LIN {X 0,Y 567.569,Z 695.919,A -85,B 0,C 180,E1 -2633.977,E2 -2633.977} C_VEL
LIN {X 0,Y 567.873,Z 675.676,A -85,B 0,C 180,E1 -2636.663,E2 -2636.663} C_VEL
LIN {X 0,Y 568.261,Z 656.786,A -85,B 0,C 180,E1 -2639.242,E2 -2639.242} C_VEL
LIN {X 0,Y 566.233,Z 647.86,A -85,B 0,C 180,E1 -2640.65,E2 -2640.65} C_VEL
LIN {X 0,Y 566.225,Z 647.758,A -85,B 0,C 180,E1 -2643.101,E2 -2643.101} C_VEL
LIN {X 0,Y 566.207,Z 647.757,A -85,B 0,C 180,E1 -2645.688,E2 -2645.688} C_VEL
LIN {X 0,Y 566.21,Z 647.762,A -85,B 0,C 180,E1 -2648.558,E2 -2648.558} C_VEL
LIN {X 0,Y 566.206,Z 647.768,A -85,B 0,C 180,E1 -2651.135,E2 -2651.135} C_VEL
LIN {X 0,Y 566.193,Z 647.762,A -85,B 0,C 180,E1 -2654.035,E2 -2654.035} C_VEL
LIN {X 0,Y 566.208,Z 647.765,A -85,B 0,C 180,E1 -2657.081,E2 -2657.081} C_VEL
LIN {X 0,Y 566.22,Z 647.768,A -85,B 0,C 180,E1 -2659.802,E2 -2659.802} C_VEL
LIN {X 0,Y 566.192,Z 647.763,A -85,B 0,C 180,E1 -2662.598,E2 -2662.598} C_VEL
LIN {X 0,Y 566.214,Z 647.758,A -85,B 0,C 180,E1 -2665.183,E2 -2665.183} C_VEL
LIN {X 0,Y 566.226,Z 647.765,A -85,B 0,C 180,E1 -2667.743,E2 -2667.743} C_VEL
LIN {X 0,Y 566.22,Z 647.758,A -85,B 0,C 180,E1 -2670.322,E2 -2670.322} C_VEL
LIN {X 0,Y 566.226,Z 647.757,A -85,B 0,C 180,E1 -2673.334,E2 -2673.334} C_VEL
LIN {X 0,Y 566.19,Z 647.766,A -85,B 0,C 180,E1 -2675.819,E2 -2675.819} C_VEL
LIN {X 0,Y 566.207,Z 647.766,A -85,B 0,C 180,E1 -2678.902,E2 -2678.902} C_VEL
LIN {X 0,Y 566.203,Z 647.763,A -85,B 0,C 180,E1 -2681.172,E2 -2681.172} C_VEL
LIN {X 0,Y 566.203,Z 647.764,A -85,B 0,C 180,E1 -2684.153,E2 -2684.153} C_VEL
LIN {X 0,Y 566.193,Z 647.766,A -85,B 0,C 180,E1 -2686.359,E2 -2686.359} C_VEL
LIN {X 0,Y 566.264,Z 647.76,A -85,B 0,C 180,E1 -2688.654,E2 -2688.654} C_VEL
LIN {X 0,Y 566.239,Z 647.758,A -85,B 0,C 180,E1 -2691.434,E2 -2691.434} C_VEL
LIN {X 0,Y 566.26,Z 647.755,A -85,B 0,C 180,E1 -2694.302,E2 -2694.302} C_VEL
LIN {X 0,Y 566.271,Z 647.754,A -85,B 0,C 180,E1 -2697.866,E2 -2697.866} C_VEL
LIN {X 0,Y 566.298,Z 647.751,A -85,B 0,C 180,E1 -2700.711,E2 -2700.711} C_VEL
LIN {X 0,Y 566.27,Z 647.752,A -85,B 0,C 180,E1 -2702.845,E2 -2702.845} C_VEL
LIN {X 0,Y 566.26,Z 647.763,A -85,B 0,C 180,E1 -2705.698,E2 -2705.698} C_VEL
LIN {X 0,Y 566.238,Z 647.757,A -85,B 0,C 180,E1 -2708.565,E2 -2708.565} C_VEL
LIN {X 0,Y 566.239,Z 647.762,A -85,B 0,C 180,E1 -2711.454,E2 -2711.454} C_VEL
LIN {X 0,Y 566.222,Z 647.762,A -85,B 0,C 180,E1 -2714.507,E2 -2714.507} C_VEL
LIN {X 0,Y 566.193,Z 647.762,A -85,B 0,C 180,E1 -2717.332,E2 -2717.332} C_VEL
LIN {X 0,Y 566.21,Z 647.769,A -85,B 0,C 180,E1 -2720.337,E2 -2720.337} C_VEL
LIN {X 0,Y 566.219,Z 647.76,A -85,B 0,C 180,E1 -2723.402,E2 -2723.402} C_VEL
LIN {X 0,Y 566.216,Z 647.762,A -85,B 0,C 180,E1 -2725.748,E2 -2725.748} C_VEL
LIN {X 0,Y 566.206,Z 647.757,A -85,B 0,C 180,E1 -2727.492,E2 -2727.492} C_VEL
LIN {X 0,Y 565.528,Z 647.847,A -85,B 0,C 180,E1 -2728.086,E2 -2728.086} C_VEL
LIN {X 0,Y 562.663,Z 648.199,A -85,B 0,C 180,E1 -2729.05,E2 -2729.05} C_VEL
LIN {X 0,Y 560.252,Z 648.499,A -85,B 0,C 180,E1 -2729.825,E2 -2729.825} C_VEL
LIN {X 0,Y 559.223,Z 648.633,A -85,B 0,C 180,E1 -2730.424,E2 -2730.424} C_VEL
LIN {X 0,Y 559.142,Z 648.641,A -85,B 0,C 180,E1 -2730.627,E2 -2730.627} C_VEL
LIN {X 0,Y 559.167,Z 648.638,A -85,B 0,C 180,E1 -2733.574,E2 -2733.574} C_VEL
LIN {X 0,Y 559.159,Z 648.636,A -85,B 0,C 180,E1 -2736.449,E2 -2736.449} C_VEL
LIN {X 0,Y 559.17,Z 648.648,A -85,B 0,C 180,E1 -2738.934,E2 -2738.934} C_VEL
LIN {X 0,Y 559.193,Z 648.637,A -85,B 0,C 180,E1 -2741.767,E2 -2741.767} C_VEL
LIN {X 0,Y 559.131,Z 648.648,A -85,B 0,C 180,E1 -2744.739,E2 -2744.739} C_VEL
LIN {X 0,Y 559.168,Z 648.642,A -85,B 0,C 180,E1 -2747.863,E2 -2747.863} C_VEL
LIN {X 0,Y 559.177,Z 648.639,A -85,B 0,C 180,E1 -2750.135,E2 -2750.135} C_VEL
LIN {X 0,Y 559.139,Z 648.645,A -85,B 0,C 180,E1 -2752.893,E2 -2752.893} C_VEL
LIN {X 0,Y 559.149,Z 648.651,A -85,B 0,C 180,E1 -2755.556,E2 -2755.556} C_VEL
LIN {X 0,Y 559.165,Z 648.643,A -85,B 0,C 180,E1 -2758.138,E2 -2758.138} C_VEL
LIN {X 0,Y 559.15,Z 648.642,A -85,B 0,C 180,E1 -2760.648,E2 -2760.648} C_VEL
LIN {X 0,Y 559.166,Z 648.641,A -85,B 0,C 180,E1 -2763.172,E2 -2763.172} C_VEL
LIN {X 0,Y 559.152,Z 648.644,A -85,B 0,C 180,E1 -2765.495,E2 -2765.495} C_VEL
LIN {X 0,Y 559.166,Z 648.643,A -85,B 0,C 180,E1 -2768.624,E2 -2768.624} C_VEL
LIN {X 0,Y 559.164,Z 648.641,A -85,B 0,C 180,E1 -2770.927,E2 -2770.927} C_VEL
LIN {X 0,Y 559.163,Z 648.644,A -85,B 0,C 180,E1 -2773.948,E2 -2773.948} C_VEL
LIN {X 0,Y 559.168,Z 648.646,A -85,B 0,C 180,E1 -2776.184,E2 -2776.184} C_VEL
LIN {X 0,Y 559.191,Z 648.639,A -85,B 0,C 180,E1 -2779.134,E2 -2779.134} C_VEL
LIN {X 0,Y 559.202,Z 648.637,A -85,B 0,C 180,E1 -2782.054,E2 -2782.054} C_VEL
LIN {X 0,Y 559.25,Z 648.638,A -85,B 0,C 180,E1 -2784.953,E2 -2784.953} C_VEL
LIN {X 0,Y 559.25,Z 648.629,A -85,B 0,C 180,E1 -2787.839,E2 -2787.839} C_VEL
LIN {X 0,Y 559.268,Z 648.633,A -85,B 0,C 180,E1 -2790.72,E2 -2790.72} C_VEL
LIN {X 0,Y 559.235,Z 648.638,A -85,B 0,C 180,E1 -2792.881,E2 -2792.881} C_VEL
LIN {X 0,Y 559.226,Z 648.635,A -85,B 0,C 180,E1 -2795.77,E2 -2795.77} C_VEL
LIN {X 0,Y 559.188,Z 648.639,A -85,B 0,C 180,E1 -2798.674,E2 -2798.674} C_VEL
LIN {X 0,Y 559.201,Z 648.644,A -85,B 0,C 180,E1 -2801.6,E2 -2801.6} C_VEL
LIN {X 0,Y 559.195,Z 648.637,A -85,B 0,C 180,E1 -2804.595,E2 -2804.595} C_VEL
LIN {X 0,Y 559.155,Z 648.649,A -85,B 0,C 180,E1 -2807.557,E2 -2807.557} C_VEL
LIN {X 0,Y 559.167,Z 648.65,A -85,B 0,C 180,E1 -2809.837,E2 -2809.837} C_VEL
LIN {X 0,Y 559.136,Z 648.65,A -85,B 0,C 180,E1 -2812.152,E2 -2812.152} C_VEL
LIN {X 0,Y 559.173,Z 648.639,A -85,B 0,C 180,E1 -2815.187,E2 -2815.187} C_VEL
LIN {X 0,Y 559.187,Z 648.641,A -85,B 0,C 180,E1 -2817.711,E2 -2817.711} C_VEL
LIN {X 0,Y 559.162,Z 648.65,A -85,B 0,C 180,E1 -2820.181,E2 -2820.181} C_VEL
LIN {X 0,Y 559.169,Z 648.644,A -85,B 0,C 180,E1 -2822.713,E2 -2822.713} C_VEL
LIN {X 0,Y 559.15,Z 648.642,A -85,B 0,C 180,E1 -2825.321,E2 -2825.321} C_VEL
LIN {X 0,Y 559.127,Z 648.647,A -85,B 0,C 180,E1 -2828.017,E2 -2828.017} C_VEL
LIN {X 0,Y 559.168,Z 648.648,A -85,B 0,C 180,E1 -2830.81,E2 -2830.81} C_VEL
LIN {X 0,Y 559.135,Z 648.643,A -85,B 0,C 180,E1 -2833.733,E2 -2833.733} C_VEL
LIN {X 0,Y 559.164,Z 648.649,A -85,B 0,C 180,E1 -2836.8,E2 -2836.8} C_VEL
LIN {X 0,Y 559.171,Z 648.646,A -85,B 0,C 180,E1 -2839.189,E2 -2839.189} C_VEL
LIN {X 0,Y 559.126,Z 648.642,A -85,B 0,C 180,E1 -2841.982,E2 -2841.982} C_VEL
LIN {X 0,Y 559.151,Z 648.637,A -85,B 0,C 180,E1 -2844.782,E2 -2844.782} C_VEL
LIN {X 0,Y 559.164,Z 648.65,A -85,B 0,C 180,E1 -2847.361,E2 -2847.361} C_VEL
LIN {X 0,Y 559.179,Z 648.631,A -85,B 0,C 180,E1 -2850.135,E2 -2850.135} C_VEL
LIN {X 0,Y 559.171,Z 648.637,A -85,B 0,C 180,E1 -2853.17,E2 -2853.17} C_VEL
LIN {X 0,Y 559.15,Z 648.649,A -85,B 0,C 180,E1 -2855.495,E2 -2855.495} C_VEL
LIN {X 0,Y 559.153,Z 648.641,A -85,B 0,C 180,E1 -2858.447,E2 -2858.447} C_VEL
LIN {X 0,Y 559.161,Z 648.639,A -85,B 0,C 180,E1 -2860.926,E2 -2860.926} C_VEL
LIN {X 0,Y 559.162,Z 648.648,A -85,B 0,C 180,E1 -2863.948,E2 -2863.948} C_VEL
LIN {X 0,Y 559.164,Z 648.644,A -85,B 0,C 180,E1 -2866.184,E2 -2866.184} C_VEL
LIN {X 0,Y 559.201,Z 648.634,A -85,B 0,C 180,E1 -2869.134,E2 -2869.134} C_VEL
LIN {X 0,Y 559.203,Z 648.638,A -85,B 0,C 180,E1 -2872.054,E2 -2872.054} C_VEL
LIN {X 0,Y 559.252,Z 648.631,A -85,B 0,C 180,E1 -2874.954,E2 -2874.954} C_VEL
LIN {X 0,Y 559.242,Z 648.627,A -85,B 0,C 180,E1 -2877.84,E2 -2877.84} C_VEL
LIN {X 0,Y 559.269,Z 648.635,A -85,B 0,C 180,E1 -2880.72,E2 -2880.72} C_VEL
LIN {X 0,Y 559.236,Z 648.637,A -85,B 0,C 180,E1 -2882.882,E2 -2882.882} C_VEL
LIN {X 0,Y 559.229,Z 648.631,A -85,B 0,C 180,E1 -2885.77,E2 -2885.77} C_VEL
LIN {X 0,Y 559.194,Z 648.636,A -85,B 0,C 180,E1 -2888.674,E2 -2888.674} C_VEL
LIN {X 0,Y 559.198,Z 648.636,A -85,B 0,C 180,E1 -2891.601,E2 -2891.601} C_VEL
LIN {X 0,Y 559.188,Z 648.636,A -85,B 0,C 180,E1 -2894.596,E2 -2894.596} C_VEL
LIN {X 0,Y 559.154,Z 648.646,A -85,B 0,C 180,E1 -2897.557,E2 -2897.557} C_VEL
LIN {X 0,Y 559.165,Z 648.643,A -85,B 0,C 180,E1 -2899.838,E2 -2899.838} C_VEL
LIN {X 0,Y 559.134,Z 648.642,A -85,B 0,C 180,E1 -2902.153,E2 -2902.153} C_VEL
LIN {X 0,Y 559.17,Z 648.642,A -85,B 0,C 180,E1 -2905.188,E2 -2905.188} C_VEL
LIN {X 0,Y 559.185,Z 648.637,A -85,B 0,C 180,E1 -2907.712,E2 -2907.712} C_VEL
LIN {X 0,Y 559.16,Z 648.643,A -85,B 0,C 180,E1 -2910.182,E2 -2910.182} C_VEL
LIN {X 0,Y 559.167,Z 648.64,A -85,B 0,C 180,E1 -2912.715,E2 -2912.715} C_VEL
LIN {X 0,Y 559.151,Z 648.637,A -85,B 0,C 180,E1 -2915.322,E2 -2915.322} C_VEL
LIN {X 0,Y 559.129,Z 648.65,A -85,B 0,C 180,E1 -2918.018,E2 -2918.018} C_VEL
LIN {X 0,Y 559.173,Z 648.636,A -85,B 0,C 180,E1 -2920.811,E2 -2920.811} C_VEL
LIN {X 0,Y 559.158,Z 648.642,A -85,B 0,C 180,E1 -2923.732,E2 -2923.732} C_VEL
LIN {X 0,Y 559.161,Z 648.647,A -85,B 0,C 180,E1 -2926.802,E2 -2926.802} C_VEL
LIN {X 0,Y 559.171,Z 648.641,A -85,B 0,C 180,E1 -2929.19,E2 -2929.19} C_VEL
LIN {X 0,Y 559.13,Z 648.644,A -85,B 0,C 180,E1 -2931.983,E2 -2931.983} C_VEL
LIN {X 0,Y 559.154,Z 648.642,A -85,B 0,C 180,E1 -2934.784,E2 -2934.784} C_VEL
LIN {X 0,Y 559.171,Z 648.628,A -85,B 0,C 180,E1 -2937.362,E2 -2937.362} C_VEL
LIN {X 0,Y 559.219,Z 648.853,A -85,B 0,C 180,E1 -2939.09,E2 -2939.09} C_VEL
LIN {X 0,Y 561.438,Z 658.244,A -85,B 0,C 180,E1 -2940.573,E2 -2940.573} C_VEL
LIN {X 0,Y 561.129,Z 674.15,A -85,B 0,C 180,E1 -2942.78,E2 -2942.78} C_VEL
LIN {X 0,Y 560.756,Z 691.767,A -85,B 0,C 180,E1 -2945.175,E2 -2945.175} C_VEL
LIN {X 0,Y 560.706,Z 696.007,A -85,B 0,C 180,E1 -2945.716,E2 -2945.716} C_VEL
LIN {X 0,Y 563.185,Z 706.581,A -85,B 0,C 180,E1 -2945.992,E2 -2945.992} C_VEL
LIN {X 0,Y 562.287,Z 897.325,A -85,B 0,C 180,E1 -2948.556,E2 -2948.556} C_VEL
LIN {X 0,Y 562.123,Z 911.373,A -85,B 0,C 180,E1 -2948.838,E2 -2948.838} C_VEL
LIN {X 0,Y 561.91,Z 924.892,A -85,B 0,C 180,E1 -2949.214,E2 -2949.214} C_VEL
LIN {X 0,Y 561.684,Z 938.18,A -85,B 0,C 180,E1 -2949.684,E2 -2949.684} C_VEL
LIN {X 0,Y 561.381,Z 951.016,A -85,B 0,C 180,E1 -2950.244,E2 -2950.244} C_VEL
LIN {X 0,Y 561.089,Z 963.63,A -85,B 0,C 180,E1 -2950.9,E2 -2950.9} C_VEL
LIN {X 0,Y 560.713,Z 977.24,A -85,B 0,C 180,E1 -2951.739,E2 -2951.739} C_VEL
LIN {X 0,Y 560.337,Z 992.413,A -85,B 0,C 180,E1 -2952.858,E2 -2952.858} C_VEL
LIN {X 0,Y 559.998,Z 1005.074,A -85,B 0,C 180,E1 -2953.973,E2 -2953.973} C_VEL
LIN {X 0,Y 559.712,Z 1015.89,A -85,B 0,C 180,E1 -2955.077,E2 -2955.077} C_VEL
LIN {X 0,Y 559.449,Z 1026.869,A -85,B 0,C 180,E1 -2956.377,E2 -2956.377} C_VEL
LIN {X 0,Y 559.241,Z 1036.211,A -85,B 0,C 180,E1 -2957.665,E2 -2957.665} C_VEL
LIN {X 0,Y 559.063,Z 1045.284,A -85,B 0,C 180,E1 -2959.131,E2 -2959.131} C_VEL
LIN {X 0,Y 558.941,Z 1052.854,A -85,B 0,C 180,E1 -2960.593,E2 -2960.593} C_VEL
LIN {X 0,Y 558.89,Z 1059.068,A -85,B 0,C 180,E1 -2962.049,E2 -2962.049} C_VEL
LIN {X 0,Y 558.841,Z 1064.1,A -85,B 0,C 180,E1 -2963.501,E2 -2963.501} C_VEL
LIN {X 0,Y 558.776,Z 1068.061,A -85,B 0,C 180,E1 -2964.949,E2 -2964.949} C_VEL
LIN {X 0,Y 558.817,Z 1070.961,A -85,B 0,C 180,E1 -2966.395,E2 -2966.395} C_VEL
LIN {X 0,Y 558.734,Z 1072.881,A -85,B 0,C 180,E1 -2967.837,E2 -2967.837} C_VEL
LIN {X 0,Y 558.738,Z 1073.833,A -85,B 0,C 180,E1 -2969.279,E2 -2969.279} C_VEL
LIN {X 0,Y 558.738,Z 1073.833,A -85,B 0,C 180,E1 -2970.721,E2 -2970.721} C_VEL
LIN {X 0,Y 558.734,Z 1072.881,A -85,B 0,C 180,E1 -2972.163,E2 -2972.163} C_VEL
LIN {X 0,Y 558.817,Z 1070.961,A -85,B 0,C 180,E1 -2973.605,E2 -2973.605} C_VEL
LIN {X 0,Y 558.776,Z 1068.061,A -85,B 0,C 180,E1 -2975.051,E2 -2975.051} C_VEL
LIN {X 0,Y 558.841,Z 1063.992,A -85,B 0,C 180,E1 -2976.535,E2 -2976.535} C_VEL
LIN {X 0,Y 558.89,Z 1059.068,A -85,B 0,C 180,E1 -2977.951,E2 -2977.951} C_VEL
LIN {X 0,Y 558.941,Z 1052.854,A -85,B 0,C 180,E1 -2979.407,E2 -2979.407} C_VEL
LIN {X 0,Y 559.115,Z 1044.27,A -85,B 0,C 180,E1 -2981.046,E2 -2981.046} C_VEL
LIN {X 0,Y 559.241,Z 1036.211,A -85,B 0,C 180,E1 -2982.335,E2 -2982.335} C_VEL
LIN {X 0,Y 559.449,Z 1026.869,A -85,B 0,C 180,E1 -2983.623,E2 -2983.623} C_VEL
LIN {X 0,Y 559.71,Z 1015.898,A -85,B 0,C 180,E1 -2984.923,E2 -2984.923} C_VEL
LIN {X 0,Y 559.975,Z 1005.074,A -85,B 0,C 180,E1 -2986.028,E2 -2986.028} C_VEL
LIN {X 0,Y 560.341,Z 991.252,A -85,B 0,C 180,E1 -2987.236,E2 -2987.236} C_VEL
LIN {X 0,Y 560.713,Z 977.24,A -85,B 0,C 180,E1 -2988.261,E2 -2988.261} C_VEL
LIN {X 0,Y 561.087,Z 963.63,A -85,B 0,C 180,E1 -2989.1,E2 -2989.1} C_VEL
LIN {X 0,Y 561.37,Z 951.016,A -85,B 0,C 180,E1 -2989.756,E2 -2989.756} C_VEL
LIN {X 0,Y 561.701,Z 936.508,A -85,B 0,C 180,E1 -2990.382,E2 -2990.382} C_VEL
LIN {X 0,Y 561.995,Z 921.141,A -85,B 0,C 180,E1 -2990.903,E2 -2990.903} C_VEL
LIN {X 0,Y 562.224,Z 902.928,A -85,B 0,C 180,E1 -2991.35,E2 -2991.35} C_VEL
LIN {X 0,Y 562.457,Z 877.103,A -85,B 0,C 180,E1 -2991.725,E2 -2991.725} C_VEL
LIN {X 0,Y 563.09,Z 705.526,A -85,B 0,C 180,E1 -2994.026,E2 -2994.026} C_VEL
LIN {X 0,Y 560.696,Z 695.906,A -85,B 0,C 180,E1 -2994.29,E2 -2994.29} C_VEL
LIN {X 0,Y 561.115,Z 676.134,A -85,B 0,C 180,E1 -2996.947,E2 -2996.947} C_VEL
LIN {X 0,Y 561.522,Z 659.701,A -85,B 0,C 180,E1 -2999.216,E2 -2999.216} C_VEL
LIN {X 0,Y 560.763,Z 655.01,A -85,B 0,C 180,E1 -2999.924,E2 -2999.924} C_VEL
LIN {X 0,Y 559.214,Z 648.775,A -85,B 0,C 180,E1 -3000.936,E2 -3000.936} C_VEL
LIN {X 0,Y 559.163,Z 648.643,A -85,B 0,C 180,E1 -3003.949,E2 -3003.949} C_VEL
LIN {X 0,Y 559.164,Z 648.63,A -85,B 0,C 180,E1 -3006.448,E2 -3006.448} C_VEL
LIN {X 0,Y 559.173,Z 648.642,A -85,B 0,C 180,E1 -3008.933,E2 -3008.933} C_VEL
LIN {X 0,Y 559.186,Z 648.642,A -85,B 0,C 180,E1 -3011.767,E2 -3011.767} C_VEL
LIN {X 0,Y 559.133,Z 648.639,A -85,B 0,C 180,E1 -3014.738,E2 -3014.738} C_VEL
LIN {X 0,Y 559.167,Z 648.644,A -85,B 0,C 180,E1 -3017.257,E2 -3017.257} C_VEL
LIN {X 0,Y 559.18,Z 648.642,A -85,B 0,C 180,E1 -3020.135,E2 -3020.135} C_VEL
LIN {X 0,Y 559.139,Z 648.641,A -85,B 0,C 180,E1 -3022.892,E2 -3022.892} C_VEL
LIN {X 0,Y 559.155,Z 648.64,A -85,B 0,C 180,E1 -3025.556,E2 -3025.556} C_VEL
LIN {X 0,Y 559.163,Z 648.647,A -85,B 0,C 180,E1 -3028.137,E2 -3028.137} C_VEL
LIN {X 0,Y 559.15,Z 648.632,A -85,B 0,C 180,E1 -3030.647,E2 -3030.647} C_VEL
LIN {X 0,Y 559.173,Z 648.635,A -85,B 0,C 180,E1 -3033.169,E2 -3033.169} C_VEL
LIN {X 0,Y 559.147,Z 648.642,A -85,B 0,C 180,E1 -3035.494,E2 -3035.494} C_VEL
LIN {X 0,Y 559.167,Z 648.648,A -85,B 0,C 180,E1 -3038.624,E2 -3038.624} C_VEL
LIN {X 0,Y 559.162,Z 648.642,A -85,B 0,C 180,E1 -3040.926,E2 -3040.926} C_VEL
LIN {X 0,Y 559.165,Z 648.639,A -85,B 0,C 180,E1 -3043.948,E2 -3043.948} C_VEL
LIN {X 0,Y 559.165,Z 648.64,A -85,B 0,C 180,E1 -3046.184,E2 -3046.184} C_VEL
LIN {X 0,Y 559.223,Z 648.639,A -85,B 0,C 180,E1 -3049.134,E2 -3049.134} C_VEL
LIN {X 0,Y 559.203,Z 648.63,A -85,B 0,C 180,E1 -3052.053,E2 -3052.053} C_VEL
LIN {X 0,Y 559.252,Z 648.635,A -85,B 0,C 180,E1 -3054.953,E2 -3054.953} C_VEL
LIN {X 0,Y 559.242,Z 648.63,A -85,B 0,C 180,E1 -3057.839,E2 -3057.839} C_VEL
LIN {X 0,Y 559.268,Z 648.627,A -85,B 0,C 180,E1 -3060.72,E2 -3060.72} C_VEL
LIN {X 0,Y 559.236,Z 648.628,A -85,B 0,C 180,E1 -3062.881,E2 -3062.881} C_VEL
LIN {X 0,Y 559.229,Z 648.638,A -85,B 0,C 180,E1 -3065.77,E2 -3065.77} C_VEL
LIN {X 0,Y 559.193,Z 648.634,A -85,B 0,C 180,E1 -3068.674,E2 -3068.674} C_VEL
LIN {X 0,Y 559.197,Z 648.642,A -85,B 0,C 180,E1 -3071.6,E2 -3071.6} C_VEL
LIN {X 0,Y 559.187,Z 648.638,A -85,B 0,C 180,E1 -3074.596,E2 -3074.596} C_VEL
LIN {X 0,Y 559.153,Z 648.641,A -85,B 0,C 180,E1 -3077.557,E2 -3077.557} C_VEL
LIN {X 0,Y 559.164,Z 648.644,A -85,B 0,C 180,E1 -3079.837,E2 -3079.837} C_VEL
LIN {X 0,Y 559.145,Z 648.649,A -85,B 0,C 180,E1 -3082.152,E2 -3082.152} C_VEL
LIN {X 0,Y 559.15,Z 648.649,A -85,B 0,C 180,E1 -3084.505,E2 -3084.505} C_VEL
LIN {X 0,Y 559.169,Z 648.636,A -85,B 0,C 180,E1 -3086.902,E2 -3086.902} C_VEL
LIN {X 0,Y 559.179,Z 648.631,A -85,B 0,C 180,E1 -3089.865,E2 -3089.865} C_VEL
LIN {X 0,Y 559.142,Z 648.641,A -85,B 0,C 180,E1 -3090.627,E2 -3090.627} C_VEL
LIN {X 0,Y 558.479,Z 648.728,A -85,B 0,C 180,E1 -3091.228,E2 -3091.228} C_VEL
LIN {X 0,Y 555.616,Z 649.084,A -85,B 0,C 180,E1 -3092.204,E2 -3092.204} C_VEL
LIN {X 0,Y 553.205,Z 649.387,A -85,B 0,C 180,E1 -3092.99,E2 -3092.99} C_VEL
LIN {X 0,Y 552.187,Z 649.508,A -85,B 0,C 180,E1 -3093.597,E2 -3093.597} C_VEL
LIN {X 0,Y 552.113,Z 649.517,A -85,B 0,C 180,E1 -3093.802,E2 -3093.802} C_VEL
LIN {X 0,Y 552.102,Z 649.517,A -85,B 0,C 180,E1 -3096.747,E2 -3096.747} C_VEL
LIN {X 0,Y 552.126,Z 649.519,A -85,B 0,C 180,E1 -3099.527,E2 -3099.527} C_VEL
LIN {X 0,Y 552.163,Z 649.516,A -85,B 0,C 180,E1 -3101.441,E2 -3101.441} C_VEL
LIN {X 0,Y 552.087,Z 649.523,A -85,B 0,C 180,E1 -3104.532,E2 -3104.532} C_VEL
LIN {X 0,Y 552.122,Z 649.523,A -85,B 0,C 180,E1 -3107.585,E2 -3107.585} C_VEL
LIN {X 0,Y 552.126,Z 649.517,A -85,B 0,C 180,E1 -3110.474,E2 -3110.474} C_VEL
LIN {X 0,Y 552.114,Z 649.526,A -85,B 0,C 180,E1 -3113.315,E2 -3113.315} C_VEL
LIN {X 0,Y 552.124,Z 649.523,A -85,B 0,C 180,E1 -3115.94,E2 -3115.94} C_VEL
LIN {X 0,Y 552.112,Z 649.519,A -85,B 0,C 180,E1 -3118.541,E2 -3118.541} C_VEL
LIN {X 0,Y 552.119,Z 649.522,A -85,B 0,C 180,E1 -3121.438,E2 -3121.438} C_VEL
LIN {X 0,Y 552.125,Z 649.521,A -85,B 0,C 180,E1 -3124.356,E2 -3124.356} C_VEL
LIN {X 0,Y 552.105,Z 649.521,A -85,B 0,C 180,E1 -3126.759,E2 -3126.759} C_VEL
LIN {X 0,Y 552.115,Z 649.518,A -85,B 0,C 180,E1 -3129.12,E2 -3129.12} C_VEL
LIN {X 0,Y 552.121,Z 649.518,A -85,B 0,C 180,E1 -3131.445,E2 -3131.445} C_VEL
LIN {X 0,Y 552.112,Z 649.52,A -85,B 0,C 180,E1 -3133.738,E2 -3133.738} C_VEL
LIN {X 0,Y 552.132,Z 649.521,A -85,B 0,C 180,E1 -3136.005,E2 -3136.005} C_VEL
LIN {X 0,Y 552.158,Z 649.517,A -85,B 0,C 180,E1 -3138.994,E2 -3138.994} C_VEL
LIN {X 0,Y 552.156,Z 649.514,A -85,B 0,C 180,E1 -3141.952,E2 -3141.952} C_VEL
LIN {X 0,Y 552.225,Z 649.513,A -85,B 0,C 180,E1 -3144.889,E2 -3144.889} C_VEL
LIN {X 0,Y 552.221,Z 649.505,A -85,B 0,C 180,E1 -3147.812,E2 -3147.812} C_VEL
LIN {X 0,Y 552.238,Z 649.509,A -85,B 0,C 180,E1 -3150.729,E2 -3150.729} C_VEL
LIN {X 0,Y 552.202,Z 649.515,A -85,B 0,C 180,E1 -3152.918,E2 -3152.918} C_VEL
LIN {X 0,Y 552.196,Z 649.51,A -85,B 0,C 180,E1 -3155.844,E2 -3155.844} C_VEL
LIN {X 0,Y 552.158,Z 649.515,A -85,B 0,C 180,E1 -3158.785,E2 -3158.785} C_VEL
LIN {X 0,Y 552.159,Z 649.519,A -85,B 0,C 180,E1 -3161.75,E2 -3161.75} C_VEL
LIN {X 0,Y 552.132,Z 649.517,A -85,B 0,C 180,E1 -3164.748,E2 -3164.748} C_VEL
LIN {X 0,Y 552.106,Z 649.528,A -85,B 0,C 180,E1 -3167.788,E2 -3167.788} C_VEL
LIN {X 0,Y 552.126,Z 649.523,A -85,B 0,C 180,E1 -3170.101,E2 -3170.101} C_VEL
LIN {X 0,Y 552.091,Z 649.524,A -85,B 0,C 180,E1 -3172.45,E2 -3172.45} C_VEL
LIN {X 0,Y 552.15,Z 649.515,A -85,B 0,C 180,E1 -3175.35,E2 -3175.35} C_VEL
LIN {X 0,Y 552.12,Z 649.527,A -85,B 0,C 180,E1 -3178.097,E2 -3178.097} C_VEL
LIN {X 0,Y 552.108,Z 649.524,A -85,B 0,C 180,E1 -3180.608,E2 -3180.608} C_VEL
LIN {X 0,Y 552.116,Z 649.519,A -85,B 0,C 180,E1 -3183.185,E2 -3183.185} C_VEL
LIN {X 0,Y 552.105,Z 649.521,A -85,B 0,C 180,E1 -3185.841,E2 -3185.841} C_VEL
LIN {X 0,Y 552.117,Z 649.521,A -85,B 0,C 180,E1 -3189.061,E2 -3189.061} C_VEL
LIN {X 0,Y 552.131,Z 649.517,A -85,B 0,C 180,E1 -3191.444,E2 -3191.444} C_VEL
LIN {X 0,Y 552.087,Z 649.528,A -85,B 0,C 180,E1 -3194.532,E2 -3194.532} C_VEL
LIN {X 0,Y 552.123,Z 649.518,A -85,B 0,C 180,E1 -3197.584,E2 -3197.584} C_VEL
LIN {X 0,Y 552.134,Z 649.516,A -85,B 0,C 180,E1 -3199.792,E2 -3199.792} C_VEL
LIN {X 0,Y 552.084,Z 649.52,A -85,B 0,C 180,E1 -3202.336,E2 -3202.336} C_VEL
LIN {X 0,Y 552.122,Z 649.516,A -85,B 0,C 180,E1 -3205.054,E2 -3205.054} C_VEL
LIN {X 0,Y 552.118,Z 649.522,A -85,B 0,C 180,E1 -3207.682,E2 -3207.682} C_VEL
LIN {X 0,Y 552.135,Z 649.507,A -85,B 0,C 180,E1 -3210.237,E2 -3210.237} C_VEL
LIN {X 0,Y 552.136,Z 649.511,A -85,B 0,C 180,E1 -3212.998,E2 -3212.998} C_VEL
LIN {X 0,Y 552.104,Z 649.522,A -85,B 0,C 180,E1 -3215.161,E2 -3215.161} C_VEL
LIN {X 0,Y 552.104,Z 649.525,A -85,B 0,C 180,E1 -3217.55,E2 -3217.55} C_VEL
LIN {X 0,Y 552.146,Z 649.513,A -85,B 0,C 180,E1 -3220.674,E2 -3220.674} C_VEL
LIN {X 0,Y 552.111,Z 649.522,A -85,B 0,C 180,E1 -3223.737,E2 -3223.737} C_VEL
LIN {X 0,Y 552.126,Z 649.525,A -85,B 0,C 180,E1 -3226.005,E2 -3226.005} C_VEL
LIN {X 0,Y 552.168,Z 649.511,A -85,B 0,C 180,E1 -3228.994,E2 -3228.994} C_VEL
LIN {X 0,Y 552.156,Z 649.515,A -85,B 0,C 180,E1 -3231.952,E2 -3231.952} C_VEL
LIN {X 0,Y 552.227,Z 649.507,A -85,B 0,C 180,E1 -3234.889,E2 -3234.889} C_VEL
LIN {X 0,Y 552.214,Z 649.502,A -85,B 0,C 180,E1 -3237.812,E2 -3237.812} C_VEL
LIN {X 0,Y 552.239,Z 649.511,A -85,B 0,C 180,E1 -3240.729,E2 -3240.729} C_VEL
LIN {X 0,Y 552.202,Z 649.513,A -85,B 0,C 180,E1 -3242.918,E2 -3242.918} C_VEL
LIN {X 0,Y 552.199,Z 649.507,A -85,B 0,C 180,E1 -3245.844,E2 -3245.844} C_VEL
LIN {X 0,Y 552.162,Z 649.513,A -85,B 0,C 180,E1 -3248.786,E2 -3248.786} C_VEL
LIN {X 0,Y 552.154,Z 649.512,A -85,B 0,C 180,E1 -3251.751,E2 -3251.751} C_VEL
LIN {X 0,Y 552.126,Z 649.518,A -85,B 0,C 180,E1 -3254.749,E2 -3254.749} C_VEL
LIN {X 0,Y 552.105,Z 649.52,A -85,B 0,C 180,E1 -3257.789,E2 -3257.789} C_VEL
LIN {X 0,Y 552.124,Z 649.518,A -85,B 0,C 180,E1 -3260.102,E2 -3260.102} C_VEL
LIN {X 0,Y 552.088,Z 649.518,A -85,B 0,C 180,E1 -3262.451,E2 -3262.451} C_VEL
LIN {X 0,Y 552.147,Z 649.519,A -85,B 0,C 180,E1 -3265.352,E2 -3265.352} C_VEL
LIN {X 0,Y 552.118,Z 649.509,A -85,B 0,C 180,E1 -3268.098,E2 -3268.098} C_VEL
LIN {X 0,Y 552.105,Z 649.517,A -85,B 0,C 180,E1 -3270.609,E2 -3270.609} C_VEL
LIN {X 0,Y 552.121,Z 649.517,A -85,B 0,C 180,E1 -3273.185,E2 -3273.185} C_VEL
LIN {X 0,Y 552.106,Z 649.519,A -85,B 0,C 180,E1 -3275.842,E2 -3275.842} C_VEL
LIN {X 0,Y 552.12,Z 649.517,A -85,B 0,C 180,E1 -3279.063,E2 -3279.063} C_VEL
LIN {X 0,Y 552.165,Z 649.506,A -85,B 0,C 180,E1 -3281.442,E2 -3281.442} C_VEL
LIN {X 0,Y 552.09,Z 649.525,A -85,B 0,C 180,E1 -3284.533,E2 -3284.533} C_VEL
LIN {X 0,Y 552.125,Z 649.517,A -85,B 0,C 180,E1 -3287.585,E2 -3287.585} C_VEL
LIN {X 0,Y 552.129,Z 649.523,A -85,B 0,C 180,E1 -3290.474,E2 -3290.474} C_VEL
LIN {X 0,Y 552.11,Z 649.507,A -85,B 0,C 180,E1 -3293.316,E2 -3293.316} C_VEL
LIN {X 0,Y 552.127,Z 649.52,A -85,B 0,C 180,E1 -3295.94,E2 -3295.94} C_VEL
LIN {X 0,Y 552.128,Z 649.643,A -85,B 0,C 180,E1 -3298.782,E2 -3298.782} C_VEL
LIN {X 0,Y 554.588,Z 659.655,A -85,B 0,C 180,E1 -3300.382,E2 -3300.382} C_VEL
LIN {X 0,Y 554.665,Z 665.531,A -85,B 0,C 180,E1 -3301.218,E2 -3301.218} C_VEL
LIN {X 0,Y 554.098,Z 687.223,A -85,B 0,C 180,E1 -3304.229,E2 -3304.229} C_VEL
LIN {X 0,Y 553.914,Z 695.92,A -85,B 0,C 180,E1 -3305.393,E2 -3305.393} C_VEL
LIN {X 0,Y 556.651,Z 707.052,A -85,B 0,C 180,E1 -3305.699,E2 -3305.699} C_VEL
LIN {X 0,Y 555.74,Z 894.458,A -85,B 0,C 180,E1 -3308.242,E2 -3308.242} C_VEL
LIN {X 0,Y 555.514,Z 909.386,A -85,B 0,C 180,E1 -3308.525,E2 -3308.525} C_VEL
LIN {X 0,Y 555.284,Z 924.13,A -85,B 0,C 180,E1 -3308.93,E2 -3308.93} C_VEL
LIN {X 0,Y 555.002,Z 937.152,A -85,B 0,C 180,E1 -3309.388,E2 -3309.388} C_VEL
LIN {X 0,Y 554.715,Z 949.907,A -85,B 0,C 180,E1 -3309.943,E2 -3309.943} C_VEL
LIN {X 0,Y 554.368,Z 961.945,A -85,B 0,C 180,E1 -3310.563,E2 -3310.563} C_VEL
LIN {X 0,Y 553.989,Z 974.377,A -85,B 0,C 180,E1 -3311.318,E2 -3311.318} C_VEL
LIN {X 0,Y 553.644,Z 986.62,A -85,B 0,C 180,E1 -3312.186,E2 -3312.186} C_VEL
LIN {X 0,Y 553.263,Z 998.97,A -85,B 0,C 180,E1 -3313.203,E2 -3313.203} C_VEL
LIN {X 0,Y 552.928,Z 1010.762,A -85,B 0,C 180,E1 -3314.33,E2 -3314.33} C_VEL
LIN {X 0,Y 552.561,Z 1023.939,A -85,B 0,C 180,E1 -3315.828,E2 -3315.828} C_VEL
LIN {X 0,Y 552.272,Z 1033.679,A -85,B 0,C 180,E1 -3317.133,E2 -3317.133} C_VEL
LIN {X 0,Y 552.125,Z 1040.927,A -85,B 0,C 180,E1 -3318.249,E2 -3318.249} C_VEL
LIN {X 0,Y 551.974,Z 1049.198,A -85,B 0,C 180,E1 -3319.732,E2 -3319.732} C_VEL
LIN {X 0,Y 551.855,Z 1056.075,A -85,B 0,C 180,E1 -3321.21,E2 -3321.21} C_VEL
LIN {X 0,Y 551.808,Z 1061.739,A -85,B 0,C 180,E1 -3322.683,E2 -3322.683} C_VEL
LIN {X 0,Y 551.77,Z 1066.23,A -85,B 0,C 180,E1 -3324.152,E2 -3324.152} C_VEL
LIN {X 0,Y 551.701,Z 1069.655,A -85,B 0,C 180,E1 -3325.617,E2 -3325.617} C_VEL
LIN {X 0,Y 551.712,Z 1072.084,A -85,B 0,C 180,E1 -3327.079,E2 -3327.079} C_VEL
LIN {X 0,Y 551.64,Z 1073.499,A -85,B 0,C 180,E1 -3328.54,E2 -3328.54} C_VEL
LIN {X 0,Y 551.636,Z 1074,A -85,B 0,C 180,E1 -3330,E2 -3330} C_VEL
LIN {X 0,Y 551.64,Z 1073.499,A -85,B 0,C 180,E1 -3331.46,E2 -3331.46} C_VEL
LIN {X 0,Y 551.712,Z 1072.084,A -85,B 0,C 180,E1 -3332.921,E2 -3332.921} C_VEL
LIN {X 0,Y 551.702,Z 1069.655,A -85,B 0,C 180,E1 -3334.383,E2 -3334.383} C_VEL
LIN {X 0,Y 551.769,Z 1066.23,A -85,B 0,C 180,E1 -3335.848,E2 -3335.848} C_VEL
LIN {X 0,Y 551.808,Z 1061.739,A -85,B 0,C 180,E1 -3337.317,E2 -3337.317} C_VEL
LIN {X 0,Y 551.855,Z 1056.075,A -85,B 0,C 180,E1 -3338.79,E2 -3338.79} C_VEL
LIN {X 0,Y 551.974,Z 1049.198,A -85,B 0,C 180,E1 -3340.268,E2 -3340.268} C_VEL
LIN {X 0,Y 552.134,Z 1040.927,A -85,B 0,C 180,E1 -3341.751,E2 -3341.751} C_VEL
LIN {X 0,Y 552.35,Z 1031.086,A -85,B 0,C 180,E1 -3343.24,E2 -3343.24} C_VEL
LIN {X 0,Y 552.662,Z 1019.263,A -85,B 0,C 180,E1 -3344.734,E2 -3344.734} C_VEL
LIN {X 0,Y 552.959,Z 1008.871,A -85,B 0,C 180,E1 -3345.858,E2 -3345.858} C_VEL
LIN {X 0,Y 553.284,Z 997.887,A -85,B 0,C 180,E1 -3346.891,E2 -3346.891} C_VEL
LIN {X 0,Y 553.678,Z 985.392,A -85,B 0,C 180,E1 -3347.908,E2 -3347.908} C_VEL
LIN {X 0,Y 554.058,Z 972.945,A -85,B 0,C 180,E1 -3348.776,E2 -3348.776} C_VEL
LIN {X 0,Y 554.433,Z 958.564,A -85,B 0,C 180,E1 -3349.628,E2 -3349.628} C_VEL
LIN {X 0,Y 554.954,Z 941.844,A -85,B 0,C 180,E1 -3350.423,E2 -3350.423} C_VEL
LIN {X 0,Y 555.233,Z 927.11,A -85,B 0,C 180,E1 -3350.975,E2 -3350.975} C_VEL
LIN {X 0,Y 555.483,Z 913.299,A -85,B 0,C 180,E1 -3351.379,E2 -3351.379} C_VEL
LIN {X 0,Y 555.659,Z 898.69,A -85,B 0,C 180,E1 -3351.688,E2 -3351.688} C_VEL
LIN {X 0,Y 556.414,Z 766.206,A -85,B 0,C 180,E1 -3353.494,E2 -3353.494} C_VEL
LIN {X 0,Y 556.652,Z 707.046,A -85,B 0,C 180,E1 -3354.301,E2 -3354.301} C_VEL
LIN {X 0,Y 553.953,Z 696.08,A -85,B 0,C 180,E1 -3354.595,E2 -3354.595} C_VEL
LIN {X 0,Y 554.317,Z 678.649,A -85,B 0,C 180,E1 -3356.952,E2 -3356.952} C_VEL
LIN {X 0,Y 554.763,Z 660.906,A -85,B 0,C 180,E1 -3359.433,E2 -3359.433} C_VEL
LIN {X 0,Y 552.783,Z 652.171,A -85,B 0,C 180,E1 -3360.778,E2 -3360.778} C_VEL
LIN {X 0,Y 552.12,Z 649.594,A -85,B 0,C 180,E1 -3361.245,E2 -3361.245} C_VEL
LIN {X 0,Y 552.134,Z 649.519,A -85,B 0,C 180,E1 -3364.171,E2 -3364.171} C_VEL
LIN {X 0,Y 552.107,Z 649.508,A -85,B 0,C 180,E1 -3366.746,E2 -3366.746} C_VEL
LIN {X 0,Y 552.129,Z 649.523,A -85,B 0,C 180,E1 -3369.526,E2 -3369.526} C_VEL
LIN {X 0,Y 552.125,Z 649.518,A -85,B 0,C 180,E1 -3372.425,E2 -3372.425} C_VEL
LIN {X 0,Y 552.093,Z 649.527,A -85,B 0,C 180,E1 -3375.562,E2 -3375.562} C_VEL
LIN {X 0,Y 552.164,Z 649.506,A -85,B 0,C 180,E1 -3378.672,E2 -3378.672} C_VEL
LIN {X 0,Y 552.114,Z 649.522,A -85,B 0,C 180,E1 -3381.411,E2 -3381.411} C_VEL
LIN {X 0,Y 552.106,Z 649.519,A -85,B 0,C 180,E1 -3384.158,E2 -3384.158} C_VEL
LIN {X 0,Y 552.121,Z 649.517,A -85,B 0,C 180,E1 -3386.815,E2 -3386.815} C_VEL
LIN {X 0,Y 552.105,Z 649.517,A -85,B 0,C 180,E1 -3389.391,E2 -3389.391} C_VEL
LIN {X 0,Y 552.118,Z 649.509,A -85,B 0,C 180,E1 -3391.902,E2 -3391.902} C_VEL
LIN {X 0,Y 552.147,Z 649.519,A -85,B 0,C 180,E1 -3394.648,E2 -3394.648} C_VEL
LIN {X 0,Y 552.088,Z 649.518,A -85,B 0,C 180,E1 -3397.549,E2 -3397.549} C_VEL
LIN {X 0,Y 552.139,Z 649.522,A -85,B 0,C 180,E1 -3400.373,E2 -3400.373} C_VEL
LIN {X 0,Y 552.148,Z 649.518,A -85,B 0,C 180,E1 -3402.977,E2 -3402.977} C_VEL
LIN {X 0,Y 552.127,Z 649.515,A -85,B 0,C 180,E1 -3406.004,E2 -3406.004} C_VEL
LIN {X 0,Y 552.183,Z 649.518,A -85,B 0,C 180,E1 -3408.994,E2 -3408.994} C_VEL
LIN {X 0,Y 552.156,Z 649.508,A -85,B 0,C 180,E1 -3411.951,E2 -3411.951} C_VEL
LIN {X 0,Y 552.227,Z 649.509,A -85,B 0,C 180,E1 -3414.889,E2 -3414.889} C_VEL
LIN {X 0,Y 552.214,Z 649.506,A -85,B 0,C 180,E1 -3417.812,E2 -3417.812} C_VEL
LIN {X 0,Y 552.237,Z 649.503,A -85,B 0,C 180,E1 -3420.729,E2 -3420.729} C_VEL
LIN {X 0,Y 552.202,Z 649.504,A -85,B 0,C 180,E1 -3422.918,E2 -3422.918} C_VEL
LIN {X 0,Y 552.199,Z 649.512,A -85,B 0,C 180,E1 -3425.844,E2 -3425.844} C_VEL
LIN {X 0,Y 552.161,Z 649.51,A -85,B 0,C 180,E1 -3428.785,E2 -3428.785} C_VEL
LIN {X 0,Y 552.153,Z 649.521,A -85,B 0,C 180,E1 -3431.75,E2 -3431.75} C_VEL
LIN {X 0,Y 552.125,Z 649.516,A -85,B 0,C 180,E1 -3434.748,E2 -3434.748} C_VEL
LIN {X 0,Y 552.104,Z 649.522,A -85,B 0,C 180,E1 -3437.788,E2 -3437.788} C_VEL
LIN {X 0,Y 552.123,Z 649.526,A -85,B 0,C 180,E1 -3440.101,E2 -3440.101} C_VEL
LIN {X 0,Y 552.104,Z 649.525,A -85,B 0,C 180,E1 -3442.45,E2 -3442.45} C_VEL
LIN {X 0,Y 552.146,Z 649.513,A -85,B 0,C 180,E1 -3445.351,E2 -3445.351} C_VEL
LIN {X 0,Y 552.117,Z 649.515,A -85,B 0,C 180,E1 -3448.097,E2 -3448.097} C_VEL
LIN {X 0,Y 552.103,Z 649.522,A -85,B 0,C 180,E1 -3450.622,E2 -3450.622} C_VEL
LIN {X 0,Y 552.119,Z 649.519,A -85,B 0,C 180,E1 -3453.185,E2 -3453.185} C_VEL
LIN {X 0,Y 552.113,Z 649.517,A -85,B 0,C 180,E1 -3453.802,E2 -3453.802} C_VEL
LIN {X 0,Y 551.479,Z 649.602,A -85,B 0,C 180,E1 -3454.411,E2 -3454.411} C_VEL
LIN {X 0,Y 548.653,Z 649.948,A -85,B 0,C 180,E1 -3455.399,E2 -3455.399} C_VEL
LIN {X 0,Y 546.227,Z 650.25,A -85,B 0,C 180,E1 -3456.194,E2 -3456.194} C_VEL
LIN {X 0,Y 545.157,Z 650.383,A -85,B 0,C 180,E1 -3456.808,E2 -3456.808} C_VEL
LIN {X 0,Y 545.055,Z 650.397,A -85,B 0,C 180,E1 -3457.016,E2 -3457.016} C_VEL
LIN {X 0,Y 545.085,Z 650.394,A -85,B 0,C 180,E1 -3460.14,E2 -3460.14} C_VEL
LIN {X 0,Y 545.059,Z 650.401,A -85,B 0,C 180,E1 -3462.698,E2 -3462.698} C_VEL
LIN {X 0,Y 545.054,Z 650.407,A -85,B 0,C 180,E1 -3465.167,E2 -3465.167} C_VEL
LIN {X 0,Y 545.074,Z 650.397,A -85,B 0,C 180,E1 -3467.898,E2 -3467.898} C_VEL
LIN {X 0,Y 545.097,Z 650.393,A -85,B 0,C 180,E1 -3470.676,E2 -3470.676} C_VEL
LIN {X 0,Y 545.053,Z 650.406,A -85,B 0,C 180,E1 -3473.622,E2 -3473.622} C_VEL
LIN {X 0,Y 545.064,Z 650.398,A -85,B 0,C 180,E1 -3476.329,E2 -3476.329} C_VEL
LIN {X 0,Y 545.064,Z 650.397,A -85,B 0,C 180,E1 -3478.953,E2 -3478.953} C_VEL
LIN {X 0,Y 545.098,Z 650.398,A -85,B 0,C 180,E1 -3481.508,E2 -3481.508} C_VEL
LIN {X 0,Y 545.089,Z 650.396,A -85,B 0,C 180,E1 -3484.491,E2 -3484.491} C_VEL
LIN {X 0,Y 545.039,Z 650.401,A -85,B 0,C 180,E1 -3487.243,E2 -3487.243} C_VEL
LIN {X 0,Y 545.115,Z 650.398,A -85,B 0,C 180,E1 -3490.415,E2 -3490.415} C_VEL
LIN {X 0,Y 545.069,Z 650.396,A -85,B 0,C 180,E1 -3493.522,E2 -3493.522} C_VEL
LIN {X 0,Y 545.091,Z 650.396,A -85,B 0,C 180,E1 -3495.82,E2 -3495.82} C_VEL
LIN {X 0,Y 545.114,Z 650.397,A -85,B 0,C 180,E1 -3498.85,E2 -3498.85} C_VEL
LIN {X 0,Y 545.126,Z 650.39,A -85,B 0,C 180,E1 -3501.847,E2 -3501.847} C_VEL
LIN {X 0,Y 545.201,Z 650.389,A -85,B 0,C 180,E1 -3504.823,E2 -3504.823} C_VEL
LIN {X 0,Y 545.193,Z 650.381,A -85,B 0,C 180,E1 -3507.784,E2 -3507.784} C_VEL
LIN {X 0,Y 545.208,Z 650.385,A -85,B 0,C 180,E1 -3510.739,E2 -3510.739} C_VEL
LIN {X 0,Y 545.169,Z 650.392,A -85,B 0,C 180,E1 -3512.956,E2 -3512.956} C_VEL
LIN {X 0,Y 545.168,Z 650.386,A -85,B 0,C 180,E1 -3515.919,E2 -3515.919} C_VEL
LIN {X 0,Y 545.117,Z 650.394,A -85,B 0,C 180,E1 -3518.9,E2 -3518.9} C_VEL
LIN {X 0,Y 545.131,Z 650.392,A -85,B 0,C 180,E1 -3521.904,E2 -3521.904} C_VEL
LIN {X 0,Y 545.081,Z 650.397,A -85,B 0,C 180,E1 -3524.943,E2 -3524.943} C_VEL
LIN {X 0,Y 545.074,Z 650.402,A -85,B 0,C 180,E1 -3528.025,E2 -3528.025} C_VEL
LIN {X 0,Y 545.09,Z 650.396,A -85,B 0,C 180,E1 -3530.372,E2 -3530.372} C_VEL
LIN {X 0,Y 545.086,Z 650.399,A -85,B 0,C 180,E1 -3533.558,E2 -3533.558} C_VEL
LIN {X 0,Y 545.074,Z 650.404,A -85,B 0,C 180,E1 -3536,E2 -3536} C_VEL
LIN {X 0,Y 545.086,Z 650.396,A -85,B 0,C 180,E1 -3538.748,E2 -3538.748} C_VEL
LIN {X 0,Y 545.072,Z 650.398,A -85,B 0,C 180,E1 -3541.682,E2 -3541.682} C_VEL
LIN {X 0,Y 545.074,Z 650.403,A -85,B 0,C 180,E1 -3544.563,E2 -3544.563} C_VEL
LIN {X 0,Y 545.033,Z 650.401,A -85,B 0,C 180,E1 -3547.303,E2 -3547.303} C_VEL
LIN {X 0,Y 545.084,Z 650.397,A -85,B 0,C 180,E1 -3550.14,E2 -3550.14} C_VEL
LIN {X 0,Y 545.069,Z 650.401,A -85,B 0,C 180,E1 -3553.106,E2 -3553.106} C_VEL
LIN {X 0,Y 545.057,Z 650.399,A -85,B 0,C 180,E1 -3556.224,E2 -3556.224} C_VEL
LIN {X 0,Y 545.114,Z 650.399,A -85,B 0,C 180,E1 -3558.889,E2 -3558.889} C_VEL
LIN {X 0,Y 545.045,Z 650.397,A -85,B 0,C 180,E1 -3561.763,E2 -3561.763} C_VEL
LIN {X 0,Y 545.056,Z 650.388,A -85,B 0,C 180,E1 -3564.534,E2 -3564.534} C_VEL
LIN {X 0,Y 545.072,Z 650.403,A -85,B 0,C 180,E1 -3567.212,E2 -3567.212} C_VEL
LIN {X 0,Y 545.091,Z 650.388,A -85,B 0,C 180,E1 -3569.813,E2 -3569.813} C_VEL
LIN {X 0,Y 545.091,Z 650.386,A -85,B 0,C 180,E1 -3572.824,E2 -3572.824} C_VEL
LIN {X 0,Y 545.049,Z 650.408,A -85,B 0,C 180,E1 -3575.631,E2 -3575.631} C_VEL
LIN {X 0,Y 545.069,Z 650.398,A -85,B 0,C 180,E1 -3578.175,E2 -3578.175} C_VEL
LIN {X 0,Y 545.109,Z 650.392,A -85,B 0,C 180,E1 -3580.415,E2 -3580.415} C_VEL
LIN {X 0,Y 545.066,Z 650.396,A -85,B 0,C 180,E1 -3583.521,E2 -3583.521} C_VEL
LIN {X 0,Y 545.084,Z 650.399,A -85,B 0,C 180,E1 -3585.82,E2 -3585.82} C_VEL
LIN {X 0,Y 545.122,Z 650.389,A -85,B 0,C 180,E1 -3588.85,E2 -3588.85} C_VEL
LIN {X 0,Y 545.125,Z 650.389,A -85,B 0,C 180,E1 -3591.847,E2 -3591.847} C_VEL
LIN {X 0,Y 545.202,Z 650.382,A -85,B 0,C 180,E1 -3594.823,E2 -3594.823} C_VEL
LIN {X 0,Y 545.185,Z 650.376,A -85,B 0,C 180,E1 -3597.784,E2 -3597.784} C_VEL
LIN {X 0,Y 545.208,Z 650.386,A -85,B 0,C 180,E1 -3600.739,E2 -3600.739} C_VEL
LIN {X 0,Y 545.168,Z 650.388,A -85,B 0,C 180,E1 -3602.956,E2 -3602.956} C_VEL
LIN {X 0,Y 545.17,Z 650.382,A -85,B 0,C 180,E1 -3605.92,E2 -3605.92} C_VEL
LIN {X 0,Y 545.119,Z 650.392,A -85,B 0,C 180,E1 -3608.9,E2 -3608.9} C_VEL
LIN {X 0,Y 545.125,Z 650.386,A -85,B 0,C 180,E1 -3611.905,E2 -3611.905} C_VEL
LIN {X 0,Y 545.075,Z 650.398,A -85,B 0,C 180,E1 -3614.944,E2 -3614.944} C_VEL
LIN {X 0,Y 545.073,Z 650.393,A -85,B 0,C 180,E1 -3618.026,E2 -3618.026} C_VEL
LIN {X 0,Y 545.089,Z 650.393,A -85,B 0,C 180,E1 -3620.372,E2 -3620.372} C_VEL
LIN {X 0,Y 545.082,Z 650.4,A -85,B 0,C 180,E1 -3623.559,E2 -3623.559} C_VEL
LIN {X 0,Y 545.08,Z 650.396,A -85,B 0,C 180,E1 -3626.001,E2 -3626.001} C_VEL
LIN {X 0,Y 545.084,Z 650.379,A -85,B 0,C 180,E1 -3628.75,E2 -3628.75} C_VEL
LIN {X 0,Y 545.069,Z 650.399,A -85,B 0,C 180,E1 -3631.683,E2 -3631.683} C_VEL
LIN {X 0,Y 545.077,Z 650.391,A -85,B 0,C 180,E1 -3634.563,E2 -3634.563} C_VEL
LIN {X 0,Y 545.034,Z 650.398,A -85,B 0,C 180,E1 -3637.304,E2 -3637.304} C_VEL
LIN {X 0,Y 545.087,Z 650.399,A -85,B 0,C 180,E1 -3640.141,E2 -3640.141} C_VEL
LIN {X 0,Y 545.062,Z 650.402,A -85,B 0,C 180,E1 -3642.698,E2 -3642.698} C_VEL
LIN {X 0,Y 545.056,Z 650.392,A -85,B 0,C 180,E1 -3645.168,E2 -3645.168} C_VEL
LIN {X 0,Y 545.077,Z 650.397,A -85,B 0,C 180,E1 -3647.898,E2 -3647.898} C_VEL
LIN {X 0,Y 545.079,Z 650.402,A -85,B 0,C 180,E1 -3650.819,E2 -3650.819} C_VEL
LIN {X 0,Y 545.051,Z 650.384,A -85,B 0,C 180,E1 -3653.621,E2 -3653.621} C_VEL
LIN {X 0,Y 545.067,Z 650.4,A -85,B 0,C 180,E1 -3656.329,E2 -3656.329} C_VEL
LIN {X 0,Y 545.123,Z 650.56,A -85,B 0,C 180,E1 -3658.509,E2 -3658.509} C_VEL
LIN {X 0,Y 547.94,Z 662.415,A -85,B 0,C 180,E1 -3660.41,E2 -3660.41} C_VEL
LIN {X 0,Y 547.535,Z 680.107,A -85,B 0,C 180,E1 -3662.893,E2 -3662.893} C_VEL
LIN {X 0,Y 547.138,Z 696.033,A -85,B 0,C 180,E1 -3665.074,E2 -3665.074} C_VEL
LIN {X 0,Y 550.21,Z 709.114,A -85,B 0,C 180,E1 -3665.425,E2 -3665.425} C_VEL
LIN {X 0,Y 549.117,Z 897.245,A -85,B 0,C 180,E1 -3668.016,E2 -3668.016} C_VEL
LIN {X 0,Y 548.868,Z 911.312,A -85,B 0,C 180,E1 -3668.302,E2 -3668.302} C_VEL
LIN {X 0,Y 548.63,Z 924.858,A -85,B 0,C 180,E1 -3668.686,E2 -3668.686} C_VEL
LIN {X 0,Y 548.304,Z 938.361,A -85,B 0,C 180,E1 -3669.175,E2 -3669.175} C_VEL
LIN {X 0,Y 547.979,Z 950.997,A -85,B 0,C 180,E1 -3669.74,E2 -3669.74} C_VEL
LIN {X 0,Y 547.63,Z 961.931,A -85,B 0,C 180,E1 -3670.314,E2 -3670.314} C_VEL
LIN {X 0,Y 547.219,Z 974.367,A -85,B 0,C 180,E1 -3671.078,E2 -3671.078} C_VEL
LIN {X 0,Y 546.852,Z 985.603,A -85,B 0,C 180,E1 -3671.878,E2 -3671.878} C_VEL
LIN {X 0,Y 546.424,Z 997.878,A -85,B 0,C 180,E1 -3672.89,E2 -3672.89} C_VEL
LIN {X 0,Y 546.072,Z 1008.862,A -85,B 0,C 180,E1 -3673.937,E2 -3673.937} C_VEL
LIN {X 0,Y 545.676,Z 1020.891,A -85,B 0,C 180,E1 -3675.264,E2 -3675.264} C_VEL
LIN {X 0,Y 545.309,Z 1032.403,A -85,B 0,C 180,E1 -3676.776,E2 -3676.776} C_VEL
LIN {X 0,Y 545.112,Z 1040.925,A -85,B 0,C 180,E1 -3678.096,E2 -3678.096} C_VEL
LIN {X 0,Y 544.96,Z 1047.299,A -85,B 0,C 180,E1 -3679.223,E2 -3679.223} C_VEL
LIN {X 0,Y 544.791,Z 1054.468,A -85,B 0,C 180,E1 -3680.721,E2 -3680.721} C_VEL
LIN {X 0,Y 544.74,Z 1060.412,A -85,B 0,C 180,E1 -3682.215,E2 -3682.215} C_VEL
LIN {X 0,Y 544.677,Z 1064.52,A -85,B 0,C 180,E1 -3683.48,E2 -3683.48} C_VEL
LIN {X 0,Y 544.619,Z 1068.05,A -85,B 0,C 180,E1 -3684.817,E2 -3684.817} C_VEL
LIN {X 0,Y 544.643,Z 1070.951,A -85,B 0,C 180,E1 -3686.301,E2 -3686.301} C_VEL
LIN {X 0,Y 544.56,Z 1072.871,A -85,B 0,C 180,E1 -3687.781,E2 -3687.781} C_VEL
LIN {X 0,Y 544.539,Z 1073.824,A -85,B 0,C 180,E1 -3689.261,E2 -3689.261} C_VEL
LIN {X 0,Y 544.539,Z 1073.824,A -85,B 0,C 180,E1 -3690.739,E2 -3690.739} C_VEL
LIN {X 0,Y 544.56,Z 1072.871,A -85,B 0,C 180,E1 -3692.219,E2 -3692.219} C_VEL
LIN {X 0,Y 544.643,Z 1070.951,A -85,B 0,C 180,E1 -3693.699,E2 -3693.699} C_VEL
LIN {X 0,Y 544.619,Z 1068.05,A -85,B 0,C 180,E1 -3695.183,E2 -3695.183} C_VEL
LIN {X 0,Y 544.69,Z 1064.093,A -85,B 0,C 180,E1 -3696.668,E2 -3696.668} C_VEL
LIN {X 0,Y 544.742,Z 1059.074,A -85,B 0,C 180,E1 -3698.159,E2 -3698.159} C_VEL
LIN {X 0,Y 544.872,Z 1051.063,A -85,B 0,C 180,E1 -3700.028,E2 -3700.028} C_VEL
LIN {X 0,Y 545.056,Z 1043.331,A -85,B 0,C 180,E1 -3701.493,E2 -3701.493} C_VEL
LIN {X 0,Y 545.251,Z 1034.942,A -85,B 0,C 180,E1 -3702.846,E2 -3702.846} C_VEL
LIN {X 0,Y 545.525,Z 1025.401,A -85,B 0,C 180,E1 -3704.168,E2 -3704.168} C_VEL
LIN {X 0,Y 545.899,Z 1014.284,A -85,B 0,C 180,E1 -3705.493,E2 -3705.493} C_VEL
LIN {X 0,Y 546.304,Z 1001.093,A -85,B 0,C 180,E1 -3706.825,E2 -3706.825} C_VEL
LIN {X 0,Y 546.736,Z 989.535,A -85,B 0,C 180,E1 -3707.819,E2 -3707.819} C_VEL
LIN {X 0,Y 547.124,Z 977.233,A -85,B 0,C 180,E1 -3708.731,E2 -3708.731} C_VEL
LIN {X 0,Y 547.535,Z 965.272,A -85,B 0,C 180,E1 -3709.495,E2 -3709.495} C_VEL
LIN {X 0,Y 547.896,Z 952.973,A -85,B 0,C 180,E1 -3710.165,E2 -3710.165} C_VEL
LIN {X 0,Y 548.27,Z 940.481,A -85,B 0,C 180,E1 -3710.739,E2 -3710.739} C_VEL
LIN {X 0,Y 548.616,Z 927.093,A -85,B 0,C 180,E1 -3711.241,E2 -3711.241} C_VEL
LIN {X 0,Y 548.864,Z 913.268,A -85,B 0,C 180,E1 -3711.649,E2 -3711.649} C_VEL
LIN {X 0,Y 549.061,Z 900.055,A -85,B 0,C 180,E1 -3711.937,E2 -3711.937} C_VEL
LIN {X 0,Y 549.365,Z 861.005,A -85,B 0,C 180,E1 -3712.494,E2 -3712.494} C_VEL
LIN {X 0,Y 550.144,Z 708.228,A -85,B 0,C 180,E1 -3714.591,E2 -3714.591} C_VEL
LIN {X 0,Y 547.134,Z 695.893,A -85,B 0,C 180,E1 -3714.935,E2 -3714.935} C_VEL
LIN {X 0,Y 547.654,Z 675.952,A -85,B 0,C 180,E1 -3717.691,E2 -3717.691} C_VEL
LIN {X 0,Y 547.951,Z 662.416,A -85,B 0,C 180,E1 -3719.589,E2 -3719.589} C_VEL
LIN {X 0,Y 545.121,Z 650.728,A -85,B 0,C 180,E1 -3721.45,E2 -3721.45} C_VEL
LIN {X 0,Y 545.074,Z 650.382,A -85,B 0,C 180,E1 -3721.682,E2 -3721.682} C_VEL
LIN {X 0,Y 545.077,Z 650.401,A -85,B 0,C 180,E1 -3724.562,E2 -3724.562} C_VEL
LIN {X 0,Y 545.034,Z 650.392,A -85,B 0,C 180,E1 -3727.303,E2 -3727.303} C_VEL
LIN {X 0,Y 545.069,Z 650.396,A -85,B 0,C 180,E1 -3730.141,E2 -3730.141} C_VEL
LIN {X 0,Y 545.08,Z 650.4,A -85,B 0,C 180,E1 -3733.105,E2 -3733.105} C_VEL
LIN {X 0,Y 545.06,Z 650.399,A -85,B 0,C 180,E1 -3736.223,E2 -3736.223} C_VEL
LIN {X 0,Y 545.116,Z 650.384,A -85,B 0,C 180,E1 -3738.889,E2 -3738.889} C_VEL
LIN {X 0,Y 545.049,Z 650.408,A -85,B 0,C 180,E1 -3741.762,E2 -3741.762} C_VEL
LIN {X 0,Y 545.058,Z 650.393,A -85,B 0,C 180,E1 -3744.533,E2 -3744.533} C_VEL
LIN {X 0,Y 545.074,Z 650.395,A -85,B 0,C 180,E1 -3747.212,E2 -3747.212} C_VEL
LIN {X 0,Y 545.093,Z 650.395,A -85,B 0,C 180,E1 -3749.812,E2 -3749.812} C_VEL
LIN {X 0,Y 545.092,Z 650.391,A -85,B 0,C 180,E1 -3752.824,E2 -3752.824} C_VEL
LIN {X 0,Y 545.043,Z 650.4,A -85,B 0,C 180,E1 -3755.63,E2 -3755.63} C_VEL
LIN {X 0,Y 545.06,Z 650.402,A -85,B 0,C 180,E1 -3758.836,E2 -3758.836} C_VEL
LIN {X 0,Y 545.074,Z 650.394,A -85,B 0,C 180,E1 -3761.195,E2 -3761.195} C_VEL
LIN {X 0,Y 545.069,Z 650.395,A -85,B 0,C 180,E1 -3763.521,E2 -3763.521} C_VEL
LIN {X 0,Y 545.086,Z 650.392,A -85,B 0,C 180,E1 -3765.82,E2 -3765.82} C_VEL
LIN {X 0,Y 545.133,Z 650.395,A -85,B 0,C 180,E1 -3768.85,E2 -3768.85} C_VEL
LIN {X 0,Y 545.126,Z 650.383,A -85,B 0,C 180,E1 -3771.847,E2 -3771.847} C_VEL
LIN {X 0,Y 545.202,Z 650.383,A -85,B 0,C 180,E1 -3774.823,E2 -3774.823} C_VEL
LIN {X 0,Y 545.186,Z 650.381,A -85,B 0,C 180,E1 -3777.783,E2 -3777.783} C_VEL
LIN {X 0,Y 545.207,Z 650.379,A -85,B 0,C 180,E1 -3780.738,E2 -3780.738} C_VEL
LIN {X 0,Y 545.168,Z 650.38,A -85,B 0,C 180,E1 -3782.956,E2 -3782.956} C_VEL
LIN {X 0,Y 545.17,Z 650.386,A -85,B 0,C 180,E1 -3785.919,E2 -3785.919} C_VEL
LIN {X 0,Y 545.118,Z 650.387,A -85,B 0,C 180,E1 -3788.9,E2 -3788.9} C_VEL
LIN {X 0,Y 545.124,Z 650.393,A -85,B 0,C 180,E1 -3791.904,E2 -3791.904} C_VEL
LIN {X 0,Y 545.074,Z 650.394,A -85,B 0,C 180,E1 -3794.944,E2 -3794.944} C_VEL
LIN {X 0,Y 545.072,Z 650.4,A -85,B 0,C 180,E1 -3798.026,E2 -3798.026} C_VEL
LIN {X 0,Y 545.088,Z 650.399,A -85,B 0,C 180,E1 -3800.372,E2 -3800.372} C_VEL
LIN {X 0,Y 545.103,Z 650.391,A -85,B 0,C 180,E1 -3803.558,E2 -3803.558} C_VEL
LIN {X 0,Y 545.078,Z 650.398,A -85,B 0,C 180,E1 -3806,E2 -3806} C_VEL
LIN {X 0,Y 545.083,Z 650.388,A -85,B 0,C 180,E1 -3808.75,E2 -3808.75} C_VEL
LIN {X 0,Y 545.067,Z 650.395,A -85,B 0,C 180,E1 -3811.683,E2 -3811.683} C_VEL
LIN {X 0,Y 545.075,Z 650.401,A -85,B 0,C 180,E1 -3814.563,E2 -3814.563} C_VEL
LIN {X 0,Y 545.055,Z 650.397,A -85,B 0,C 180,E1 -3817.016,E2 -3817.016} C_VEL
LIN {X 0,Y 544.351,Z 650.487,A -85,B 0,C 180,E1 -3817.633,E2 -3817.633} C_VEL
LIN {X 0,Y 541.497,Z 650.844,A -85,B 0,C 180,E1 -3818.634,E2 -3818.634} C_VEL
LIN {X 0,Y 539.12,Z 651.14,A -85,B 0,C 180,E1 -3819.439,E2 -3819.439} C_VEL
LIN {X 0,Y 538.115,Z 651.263,A -85,B 0,C 180,E1 -3820.062,E2 -3820.062} C_VEL
LIN {X 0,Y 538.04,Z 651.273,A -85,B 0,C 180,E1 -3820.272,E2 -3820.272} C_VEL
LIN {X 0,Y 538.026,Z 651.282,A -85,B 0,C 180,E1 -3822.989,E2 -3822.989} C_VEL
LIN {X 0,Y 538.021,Z 651.275,A -85,B 0,C 180,E1 -3825.926,E2 -3825.926} C_VEL
LIN {X 0,Y 538.07,Z 651.276,A -85,B 0,C 180,E1 -3829.249,E2 -3829.249} C_VEL
LIN {X 0,Y 537.986,Z 651.28,A -85,B 0,C 180,E1 -3832.123,E2 -3832.123} C_VEL
LIN {X 0,Y 538.012,Z 651.277,A -85,B 0,C 180,E1 -3834.918,E2 -3834.918} C_VEL
LIN {X 0,Y 538.025,Z 651.282,A -85,B 0,C 180,E1 -3837.619,E2 -3837.619} C_VEL
LIN {X 0,Y 538.037,Z 651.276,A -85,B 0,C 180,E1 -3840.241,E2 -3840.241} C_VEL
LIN {X 0,Y 538.061,Z 651.27,A -85,B 0,C 180,E1 -3842.797,E2 -3842.797} C_VEL
LIN {X 0,Y 538.043,Z 651.273,A -85,B 0,C 180,E1 -3845.293,E2 -3845.293} C_VEL
LIN {X 0,Y 538.01,Z 651.284,A -85,B 0,C 180,E1 -3848.042,E2 -3848.042} C_VEL
LIN {X 0,Y 538.033,Z 651.274,A -85,B 0,C 180,E1 -3850.94,E2 -3850.94} C_VEL
LIN {X 0,Y 538.02,Z 651.274,A -85,B 0,C 180,E1 -3853.299,E2 -3853.299} C_VEL
LIN {X 0,Y 538.06,Z 651.271,A -85,B 0,C 180,E1 -3855.631,E2 -3855.631} C_VEL
LIN {X 0,Y 538.073,Z 651.276,A -85,B 0,C 180,E1 -3858.702,E2 -3858.702} C_VEL
LIN {X 0,Y 538.083,Z 651.267,A -85,B 0,C 180,E1 -3861.74,E2 -3861.74} C_VEL
LIN {X 0,Y 538.158,Z 651.266,A -85,B 0,C 180,E1 -3864.755,E2 -3864.755} C_VEL
LIN {X 0,Y 538.165,Z 651.257,A -85,B 0,C 180,E1 -3867.755,E2 -3867.755} C_VEL
LIN {X 0,Y 538.179,Z 651.262,A -85,B 0,C 180,E1 -3870.748,E2 -3870.748} C_VEL
LIN {X 0,Y 538.135,Z 651.269,A -85,B 0,C 180,E1 -3872.994,E2 -3872.994} C_VEL
LIN {X 0,Y 538.121,Z 651.263,A -85,B 0,C 180,E1 -3875.997,E2 -3875.997} C_VEL
LIN {X 0,Y 538.068,Z 651.274,A -85,B 0,C 180,E1 -3879.017,E2 -3879.017} C_VEL
LIN {X 0,Y 538.079,Z 651.269,A -85,B 0,C 180,E1 -3882.062,E2 -3882.062} C_VEL
LIN {X 0,Y 538.041,Z 651.276,A -85,B 0,C 180,E1 -3885.143,E2 -3885.143} C_VEL
LIN {X 0,Y 538.027,Z 651.277,A -85,B 0,C 180,E1 -3888.27,E2 -3888.27} C_VEL
LIN {X 0,Y 538.034,Z 651.273,A -85,B 0,C 180,E1 -3890.651,E2 -3890.651} C_VEL
LIN {X 0,Y 538.019,Z 651.283,A -85,B 0,C 180,E1 -3893.887,E2 -3893.887} C_VEL
LIN {X 0,Y 538.037,Z 651.278,A -85,B 0,C 180,E1 -3896.366,E2 -3896.366} C_VEL
LIN {X 0,Y 538.05,Z 651.272,A -85,B 0,C 180,E1 -3898.938,E2 -3898.938} C_VEL
LIN {X 0,Y 538.021,Z 651.278,A -85,B 0,C 180,E1 -3901.89,E2 -3901.89} C_VEL
LIN {X 0,Y 538.024,Z 651.281,A -85,B 0,C 180,E1 -3904.62,E2 -3904.62} C_VEL
LIN {X 0,Y 538.002,Z 651.278,A -85,B 0,C 180,E1 -3907.17,E2 -3907.17} C_VEL
LIN {X 0,Y 538.046,Z 651.271,A -85,B 0,C 180,E1 -3909.794,E2 -3909.794} C_VEL
LIN {X 0,Y 538.011,Z 651.284,A -85,B 0,C 180,E1 -3912.785,E2 -3912.785} C_VEL
LIN {X 0,Y 538.023,Z 651.279,A -85,B 0,C 180,E1 -3915.14,E2 -3915.14} C_VEL
LIN {X 0,Y 538.051,Z 651.271,A -85,B 0,C 180,E1 -3918.229,E2 -3918.229} C_VEL
LIN {X 0,Y 538.007,Z 651.282,A -85,B 0,C 180,E1 -3921.17,E2 -3921.17} C_VEL
LIN {X 0,Y 538.02,Z 651.263,A -85,B 0,C 180,E1 -3924.083,E2 -3924.083} C_VEL
LIN {X 0,Y 538.025,Z 651.274,A -85,B 0,C 180,E1 -3926.728,E2 -3926.728} C_VEL
LIN {X 0,Y 538.027,Z 651.271,A -85,B 0,C 180,E1 -3929.554,E2 -3929.554} C_VEL
LIN {X 0,Y 538.038,Z 651.267,A -85,B 0,C 180,E1 -3931.95,E2 -3931.95} C_VEL
LIN {X 0,Y 538.065,Z 651.268,A -85,B 0,C 180,E1 -3934.467,E2 -3934.467} C_VEL
LIN {X 0,Y 538.033,Z 651.271,A -85,B 0,C 180,E1 -3936.929,E2 -3936.929} C_VEL
LIN {X 0,Y 538.067,Z 651.272,A -85,B 0,C 180,E1 -3940.148,E2 -3940.148} C_VEL
LIN {X 0,Y 538.017,Z 651.272,A -85,B 0,C 180,E1 -3943.299,E2 -3943.299} C_VEL
LIN {X 0,Y 538.052,Z 651.272,A -85,B 0,C 180,E1 -3945.631,E2 -3945.631} C_VEL
LIN {X 0,Y 538.078,Z 651.268,A -85,B 0,C 180,E1 -3948.702,E2 -3948.702} C_VEL
LIN {X 0,Y 538.081,Z 651.265,A -85,B 0,C 180,E1 -3951.74,E2 -3951.74} C_VEL
LIN {X 0,Y 538.178,Z 651.258,A -85,B 0,C 180,E1 -3954.755,E2 -3954.755} C_VEL
LIN {X 0,Y 538.157,Z 651.251,A -85,B 0,C 180,E1 -3957.755,E2 -3957.755} C_VEL
LIN {X 0,Y 538.177,Z 651.261,A -85,B 0,C 180,E1 -3960.748,E2 -3960.748} C_VEL
LIN {X 0,Y 538.134,Z 651.263,A -85,B 0,C 180,E1 -3962.995,E2 -3962.995} C_VEL
LIN {X 0,Y 538.124,Z 651.26,A -85,B 0,C 180,E1 -3965.997,E2 -3965.997} C_VEL
LIN {X 0,Y 538.068,Z 651.272,A -85,B 0,C 180,E1 -3969.018,E2 -3969.018} C_VEL
LIN {X 0,Y 538.073,Z 651.264,A -85,B 0,C 180,E1 -3972.063,E2 -3972.063} C_VEL
LIN {X 0,Y 538.035,Z 651.279,A -85,B 0,C 180,E1 -3975.144,E2 -3975.144} C_VEL
LIN {X 0,Y 538.025,Z 651.27,A -85,B 0,C 180,E1 -3978.27,E2 -3978.27} C_VEL
LIN {X 0,Y 538.033,Z 651.272,A -85,B 0,C 180,E1 -3980.652,E2 -3980.652} C_VEL
LIN {X 0,Y 538.014,Z 651.28,A -85,B 0,C 180,E1 -3983.888,E2 -3983.888} C_VEL
LIN {X 0,Y 538.041,Z 651.268,A -85,B 0,C 180,E1 -3986.367,E2 -3986.367} C_VEL
LIN {X 0,Y 538.047,Z 651.254,A -85,B 0,C 180,E1 -3988.939,E2 -3988.939} C_VEL
LIN {X 0,Y 538.019,Z 651.281,A -85,B 0,C 180,E1 -3991.891,E2 -3991.891} C_VEL
LIN {X 0,Y 538.027,Z 651.268,A -85,B 0,C 180,E1 -3994.622,E2 -3994.622} C_VEL
LIN {X 0,Y 538.003,Z 651.273,A -85,B 0,C 180,E1 -3997.172,E2 -3997.172} C_VEL
LIN {X 0,Y 538.048,Z 651.274,A -85,B 0,C 180,E1 -3999.795,E2 -3999.795} C_VEL
LIN {X 0,Y 538.019,Z 651.279,A -85,B 0,C 180,E1 -4002.786,E2 -4002.786} C_VEL
LIN {X 0,Y 538.022,Z 651.269,A -85,B 0,C 180,E1 -4005.926,E2 -4005.926} C_VEL
LIN {X 0,Y 538.046,Z 651.272,A -85,B 0,C 180,E1 -4009.225,E2 -4009.225} C_VEL
LIN {X 0,Y 537.989,Z 651.278,A -85,B 0,C 180,E1 -4012.123,E2 -4012.123} C_VEL
LIN {X 0,Y 538.015,Z 651.275,A -85,B 0,C 180,E1 -4014.918,E2 -4014.918} C_VEL
LIN {X 0,Y 538.028,Z 651.255,A -85,B 0,C 180,E1 -4017.619,E2 -4017.619} C_VEL
LIN {X 0,Y 538.063,Z 651.473,A -85,B 0,C 180,E1 -4018.213,E2 -4018.213} C_VEL
LIN {X 0,Y 541.046,Z 663.677,A -85,B 0,C 180,E1 -4020.209,E2 -4020.209} C_VEL
LIN {X 0,Y 541.072,Z 669.629,A -85,B 0,C 180,E1 -4021.066,E2 -4021.066} C_VEL
LIN {X 0,Y 540.435,Z 691.875,A -85,B 0,C 180,E1 -4024.19,E2 -4024.19} C_VEL
LIN {X 0,Y 540.35,Z 696.024,A -85,B 0,C 180,E1 -4024.738,E2 -4024.738} C_VEL
LIN {X 0,Y 543.734,Z 709.719,A -85,B 0,C 180,E1 -4025.121,E2 -4025.121} C_VEL
LIN {X 0,Y 542.594,Z 894.396,A -85,B 0,C 180,E1 -4027.687,E2 -4027.687} C_VEL
LIN {X 0,Y 542.314,Z 909.326,A -85,B 0,C 180,E1 -4027.976,E2 -4027.976} C_VEL
LIN {X 0,Y 542.061,Z 923.352,A -85,B 0,C 180,E1 -4028.365,E2 -4028.365} C_VEL
LIN {X 0,Y 541.726,Z 935.273,A -85,B 0,C 180,E1 -4028.782,E2 -4028.782} C_VEL
LIN {X 0,Y 541.324,Z 949.127,A -85,B 0,C 180,E1 -4029.387,E2 -4029.387} C_VEL
LIN {X 0,Y 540.875,Z 961.917,A -85,B 0,C 180,E1 -4030.058,E2 -4030.058} C_VEL
LIN {X 0,Y 540.467,Z 974.358,A -85,B 0,C 180,E1 -4030.832,E2 -4030.832} C_VEL
LIN {X 0,Y 540.035,Z 985.121,A -85,B 0,C 180,E1 -4031.604,E2 -4031.604} C_VEL
LIN {X 0,Y 539.583,Z 996.787,A -85,B 0,C 180,E1 -4032.569,E2 -4032.569} C_VEL
LIN {X 0,Y 539.187,Z 1006.959,A -85,B 0,C 180,E1 -4033.531,E2 -4033.531} C_VEL
LIN {X 0,Y 538.822,Z 1017.597,A -85,B 0,C 180,E1 -4034.685,E2 -4034.685} C_VEL
LIN {X 0,Y 538.487,Z 1026.848,A -85,B 0,C 180,E1 -4035.835,E2 -4035.835} C_VEL
LIN {X 0,Y 538.196,Z 1036.204,A -85,B 0,C 180,E1 -4037.174,E2 -4037.174} C_VEL
LIN {X 0,Y 537.935,Z 1046.307,A -85,B 0,C 180,E1 -4038.89,E2 -4038.89} C_VEL
LIN {X 0,Y 537.743,Z 1052.848,A -85,B 0,C 180,E1 -4040.218,E2 -4040.218} C_VEL
LIN {X 0,Y 537.668,Z 1059.073,A -85,B 0,C 180,E1 -4041.733,E2 -4041.733} C_VEL
LIN {X 0,Y 537.614,Z 1064.089,A -85,B 0,C 180,E1 -4043.244,E2 -4043.244} C_VEL
LIN {X 0,Y 537.544,Z 1068.044,A -85,B 0,C 180,E1 -4044.749,E2 -4044.749} C_VEL
LIN {X 0,Y 537.559,Z 1070.947,A -85,B 0,C 180,E1 -4046.252,E2 -4046.252} C_VEL
LIN {X 0,Y 537.479,Z 1072.866,A -85,B 0,C 180,E1 -4047.752,E2 -4047.752} C_VEL
LIN {X 0,Y 537.439,Z 1073.819,A -85,B 0,C 180,E1 -4049.251,E2 -4049.251} C_VEL
LIN {X 0,Y 537.439,Z 1073.819,A -85,B 0,C 180,E1 -4050.749,E2 -4050.749} C_VEL
LIN {X 0,Y 537.479,Z 1072.866,A -85,B 0,C 180,E1 -4052.248,E2 -4052.248} C_VEL
LIN {X 0,Y 537.559,Z 1070.947,A -85,B 0,C 180,E1 -4053.748,E2 -4053.748} C_VEL
LIN {X 0,Y 537.544,Z 1068.044,A -85,B 0,C 180,E1 -4055.251,E2 -4055.251} C_VEL
LIN {X 0,Y 537.614,Z 1064.089,A -85,B 0,C 180,E1 -4056.756,E2 -4056.756} C_VEL
LIN {X 0,Y 537.668,Z 1059.073,A -85,B 0,C 180,E1 -4058.267,E2 -4058.267} C_VEL
LIN {X 0,Y 537.832,Z 1051.065,A -85,B 0,C 180,E1 -4060.16,E2 -4060.16} C_VEL
LIN {X 0,Y 538.049,Z 1042.834,A -85,B 0,C 180,E1 -4061.73,E2 -4061.73} C_VEL
LIN {X 0,Y 538.221,Z 1034.935,A -85,B 0,C 180,E1 -4063.017,E2 -4063.017} C_VEL
LIN {X 0,Y 538.573,Z 1025.393,A -85,B 0,C 180,E1 -4064.355,E2 -4064.355} C_VEL
LIN {X 0,Y 538.913,Z 1015.939,A -85,B 0,C 180,E1 -4065.505,E2 -4065.505} C_VEL
LIN {X 0,Y 539.267,Z 1005.064,A -85,B 0,C 180,E1 -4066.661,E2 -4066.661} C_VEL
LIN {X 0,Y 539.875,Z 990.32,A -85,B 0,C 180,E1 -4067.99,E2 -4067.99} C_VEL
LIN {X 0,Y 540.344,Z 977.223,A -85,B 0,C 180,E1 -4068.975,E2 -4068.975} C_VEL
LIN {X 0,Y 540.788,Z 965.258,A -85,B 0,C 180,E1 -4069.748,E2 -4069.748} C_VEL
LIN {X 0,Y 541.197,Z 952.963,A -85,B 0,C 180,E1 -4070.426,E2 -4070.426} C_VEL
LIN {X 0,Y 541.603,Z 940.949,A -85,B 0,C 180,E1 -4070.986,E2 -4070.986} C_VEL
LIN {X 0,Y 542.012,Z 927.076,A -85,B 0,C 180,E1 -4071.512,E2 -4071.512} C_VEL
LIN {X 0,Y 542.252,Z 913.238,A -85,B 0,C 180,E1 -4071.927,E2 -4071.927} C_VEL
LIN {X 0,Y 542.474,Z 900.016,A -85,B 0,C 180,E1 -4072.218,E2 -4072.218} C_VEL
LIN {X 0,Y 542.818,Z 862.794,A -85,B 0,C 180,E1 -4072.755,E2 -4072.755} C_VEL
LIN {X 0,Y 543.693,Z 709.539,A -85,B 0,C 180,E1 -4074.884,E2 -4074.884} C_VEL
LIN {X 0,Y 540.373,Z 696.128,A -85,B 0,C 180,E1 -4075.254,E2 -4075.254} C_VEL
LIN {X 0,Y 540.534,Z 688.852,A -85,B 0,C 180,E1 -4076.235,E2 -4076.235} C_VEL
LIN {X 0,Y 541.201,Z 666.345,A -85,B 0,C 180,E1 -4079.398,E2 -4079.398} C_VEL
LIN {X 0,Y 540.773,Z 662.183,A -85,B 0,C 180,E1 -4080.023,E2 -4080.023} C_VEL
LIN {X 0,Y 538.063,Z 651.476,A -85,B 0,C 180,E1 -4081.787,E2 -4081.787} C_VEL
LIN {X 0,Y 538.027,Z 651.28,A -85,B 0,C 180,E1 -4084.62,E2 -4084.62} C_VEL
LIN {X 0,Y 538.003,Z 651.264,A -85,B 0,C 180,E1 -4087.17,E2 -4087.17} C_VEL
LIN {X 0,Y 538.024,Z 651.276,A -85,B 0,C 180,E1 -4089.796,E2 -4089.796} C_VEL
LIN {X 0,Y 538.018,Z 651.277,A -85,B 0,C 180,E1 -4092.785,E2 -4092.785} C_VEL
LIN {X 0,Y 538.024,Z 651.279,A -85,B 0,C 180,E1 -4095.925,E2 -4095.925} C_VEL
LIN {X 0,Y 538.074,Z 651.263,A -85,B 0,C 180,E1 -4099.248,E2 -4099.248} C_VEL
LIN {X 0,Y 537.988,Z 651.281,A -85,B 0,C 180,E1 -4102.122,E2 -4102.122} C_VEL
LIN {X 0,Y 538.014,Z 651.268,A -85,B 0,C 180,E1 -4104.917,E2 -4104.917} C_VEL
LIN {X 0,Y 538.024,Z 651.277,A -85,B 0,C 180,E1 -4107.618,E2 -4107.618} C_VEL
LIN {X 0,Y 538.034,Z 651.265,A -85,B 0,C 180,E1 -4110.24,E2 -4110.24} C_VEL
LIN {X 0,Y 538.062,Z 651.267,A -85,B 0,C 180,E1 -4112.796,E2 -4112.796} C_VEL
LIN {X 0,Y 538.04,Z 651.271,A -85,B 0,C 180,E1 -4115.292,E2 -4115.292} C_VEL
LIN {X 0,Y 538.005,Z 651.275,A -85,B 0,C 180,E1 -4118.041,E2 -4118.041} C_VEL
LIN {X 0,Y 538.031,Z 651.274,A -85,B 0,C 180,E1 -4120.94,E2 -4120.94} C_VEL
LIN {X 0,Y 538.019,Z 651.275,A -85,B 0,C 180,E1 -4123.299,E2 -4123.299} C_VEL
LIN {X 0,Y 538.054,Z 651.268,A -85,B 0,C 180,E1 -4125.63,E2 -4125.63} C_VEL
LIN {X 0,Y 538.087,Z 651.27,A -85,B 0,C 180,E1 -4128.702,E2 -4128.702} C_VEL
LIN {X 0,Y 538.082,Z 651.261,A -85,B 0,C 180,E1 -4131.739,E2 -4131.739} C_VEL
LIN {X 0,Y 538.178,Z 651.257,A -85,B 0,C 180,E1 -4134.755,E2 -4134.755} C_VEL
LIN {X 0,Y 538.158,Z 651.257,A -85,B 0,C 180,E1 -4137.755,E2 -4137.755} C_VEL
LIN {X 0,Y 538.177,Z 651.255,A -85,B 0,C 180,E1 -4140.748,E2 -4140.748} C_VEL
LIN {X 0,Y 538.134,Z 651.256,A -85,B 0,C 180,E1 -4142.994,E2 -4142.994} C_VEL
LIN {X 0,Y 538.123,Z 651.263,A -85,B 0,C 180,E1 -4145.997,E2 -4145.997} C_VEL
LIN {X 0,Y 538.067,Z 651.266,A -85,B 0,C 180,E1 -4149.017,E2 -4149.017} C_VEL
LIN {X 0,Y 538.072,Z 651.268,A -85,B 0,C 180,E1 -4152.062,E2 -4152.062} C_VEL
LIN {X 0,Y 538.034,Z 651.272,A -85,B 0,C 180,E1 -4155.144,E2 -4155.144} C_VEL
LIN {X 0,Y 538.024,Z 651.28,A -85,B 0,C 180,E1 -4158.27,E2 -4158.27} C_VEL
LIN {X 0,Y 538.032,Z 651.274,A -85,B 0,C 180,E1 -4160.651,E2 -4160.651} C_VEL
LIN {X 0,Y 538.033,Z 651.271,A -85,B 0,C 180,E1 -4163.071,E2 -4163.071} C_VEL
LIN {X 0,Y 538.038,Z 651.272,A -85,B 0,C 180,E1 -4165.674,E2 -4165.674} C_VEL
LIN {X 0,Y 538.038,Z 651.267,A -85,B 0,C 180,E1 -4168.05,E2 -4168.05} C_VEL
LIN {X 0,Y 538.018,Z 651.276,A -85,B 0,C 180,E1 -4170.627,E2 -4170.627} C_VEL
LIN {X 0,Y 538.034,Z 651.273,A -85,B 0,C 180,E1 -4173.283,E2 -4173.283} C_VEL
LIN {X 0,Y 538.018,Z 651.263,A -85,B 0,C 180,E1 -4176.002,E2 -4176.002} C_VEL
LIN {X 0,Y 538.007,Z 651.282,A -85,B 0,C 180,E1 -4178.83,E2 -4178.83} C_VEL
LIN {X 0,Y 538.04,Z 651.273,A -85,B 0,C 180,E1 -4180.272,E2 -4180.272} C_VEL
LIN {X 0,Y 537.389,Z 651.361,A -85,B 0,C 180,E1 -4180.897,E2 -4180.897} C_VEL
LIN {X 0,Y 534.53,Z 651.719,A -85,B 0,C 180,E1 -4181.912,E2 -4181.912} C_VEL
LIN {X 0,Y 532.097,Z 652.022,A -85,B 0,C 180,E1 -4182.729,E2 -4182.729} C_VEL
LIN {X 0,Y 531.045,Z 652.15,A -85,B 0,C 180,E1 -4183.36,E2 -4183.36} C_VEL
LIN {X 0,Y 530.956,Z 652.158,A -85,B 0,C 180,E1 -4183.573,E2 -4183.573} C_VEL
LIN {X 0,Y 530.956,Z 652.155,A -85,B 0,C 180,E1 -4186.506,E2 -4186.506} C_VEL
LIN {X 0,Y 531.018,Z 652.153,A -85,B 0,C 180,E1 -4189.572,E2 -4189.572} C_VEL
LIN {X 0,Y 530.962,Z 652.154,A -85,B 0,C 180,E1 -4192.577,E2 -4192.577} C_VEL
LIN {X 0,Y 530.994,Z 652.155,A -85,B 0,C 180,E1 -4195.312,E2 -4195.312} C_VEL
LIN {X 0,Y 530.976,Z 652.157,A -85,B 0,C 180,E1 -4198.033,E2 -4198.033} C_VEL
LIN {X 0,Y 530.99,Z 652.151,A -85,B 0,C 180,E1 -4200.873,E2 -4200.873} C_VEL
LIN {X 0,Y 531.001,Z 652.151,A -85,B 0,C 180,E1 -4203.257,E2 -4203.257} C_VEL
LIN {X 0,Y 530.992,Z 652.158,A -85,B 0,C 180,E1 -4205.958,E2 -4205.958} C_VEL
LIN {X 0,Y 530.995,Z 652.15,A -85,B 0,C 180,E1 -4209.062,E2 -4209.062} C_VEL
LIN {X 0,Y 531.012,Z 652.156,A -85,B 0,C 180,E1 -4212.278,E2 -4212.278} C_VEL
LIN {X 0,Y 531.015,Z 652.148,A -85,B 0,C 180,E1 -4215.436,E2 -4215.436} C_VEL
LIN {X 0,Y 531.033,Z 652.153,A -85,B 0,C 180,E1 -4218.55,E2 -4218.55} C_VEL
LIN {X 0,Y 531.053,Z 652.143,A -85,B 0,C 180,E1 -4221.63,E2 -4221.63} C_VEL
LIN {X 0,Y 531.118,Z 652.142,A -85,B 0,C 180,E1 -4224.685,E2 -4224.685} C_VEL
LIN {X 0,Y 531.137,Z 652.133,A -85,B 0,C 180,E1 -4227.725,E2 -4227.725} C_VEL
LIN {X 0,Y 531.149,Z 652.137,A -85,B 0,C 180,E1 -4230.758,E2 -4230.758} C_VEL
LIN {X 0,Y 531.102,Z 652.145,A -85,B 0,C 180,E1 -4233.034,E2 -4233.034} C_VEL
LIN {X 0,Y 531.081,Z 652.14,A -85,B 0,C 180,E1 -4236.077,E2 -4236.077} C_VEL
LIN {X 0,Y 531.028,Z 652.152,A -85,B 0,C 180,E1 -4239.138,E2 -4239.138} C_VEL
LIN {X 0,Y 531.036,Z 652.146,A -85,B 0,C 180,E1 -4242.225,E2 -4242.225} C_VEL
LIN {X 0,Y 530.991,Z 652.157,A -85,B 0,C 180,E1 -4245.349,E2 -4245.349} C_VEL
LIN {X 0,Y 530.986,Z 652.152,A -85,B 0,C 180,E1 -4248.521,E2 -4248.521} C_VEL
LIN {X 0,Y 530.995,Z 652.15,A -85,B 0,C 180,E1 -4250.938,E2 -4250.938} C_VEL
LIN {X 0,Y 530.975,Z 652.158,A -85,B 0,C 180,E1 -4254.224,E2 -4254.224} C_VEL
LIN {X 0,Y 531.001,Z 652.151,A -85,B 0,C 180,E1 -4256.743,E2 -4256.743} C_VEL
LIN {X 0,Y 530.994,Z 652.15,A -85,B 0,C 180,E1 -4259.321,E2 -4259.321} C_VEL
LIN {X 0,Y 530.974,Z 652.159,A -85,B 0,C 180,E1 -4262.103,E2 -4262.103} C_VEL
LIN {X 0,Y 530.981,Z 652.155,A -85,B 0,C 180,E1 -4264.854,E2 -4264.854} C_VEL
LIN {X 0,Y 530.959,Z 652.154,A -85,B 0,C 180,E1 -4267.507,E2 -4267.507} C_VEL
LIN {X 0,Y 531.018,Z 652.153,A -85,B 0,C 180,E1 -4270.428,E2 -4270.428} C_VEL
LIN {X 0,Y 530.956,Z 652.155,A -85,B 0,C 180,E1 -4273.494,E2 -4273.494} C_VEL
LIN {X 0,Y 530.959,Z 652.158,A -85,B 0,C 180,E1 -4276.505,E2 -4276.505} C_VEL
LIN {X 0,Y 531,Z 652.151,A -85,B 0,C 180,E1 -4279.569,E2 -4279.569} C_VEL
LIN {X 0,Y 530.959,Z 652.153,A -85,B 0,C 180,E1 -4282.576,E2 -4282.576} C_VEL
LIN {X 0,Y 530.994,Z 652.149,A -85,B 0,C 180,E1 -4285.311,E2 -4285.311} C_VEL
LIN {X 0,Y 530.972,Z 652.152,A -85,B 0,C 180,E1 -4288.033,E2 -4288.033} C_VEL
LIN {X 0,Y 530.996,Z 652.14,A -85,B 0,C 180,E1 -4290.87,E2 -4290.87} C_VEL
LIN {X 0,Y 531.001,Z 652.144,A -85,B 0,C 180,E1 -4293.257,E2 -4293.257} C_VEL
LIN {X 0,Y 530.996,Z 652.153,A -85,B 0,C 180,E1 -4295.955,E2 -4295.955} C_VEL
LIN {X 0,Y 530.994,Z 652.148,A -85,B 0,C 180,E1 -4299.062,E2 -4299.062} C_VEL
LIN {X 0,Y 531.005,Z 652.149,A -85,B 0,C 180,E1 -4302.278,E2 -4302.278} C_VEL
LIN {X 0,Y 531.007,Z 652.148,A -85,B 0,C 180,E1 -4305.436,E2 -4305.436} C_VEL
LIN {X 0,Y 531.035,Z 652.147,A -85,B 0,C 180,E1 -4308.55,E2 -4308.55} C_VEL
LIN {X 0,Y 531.05,Z 652.14,A -85,B 0,C 180,E1 -4311.63,E2 -4311.63} C_VEL
LIN {X 0,Y 531.134,Z 652.137,A -85,B 0,C 180,E1 -4314.686,E2 -4314.686} C_VEL
LIN {X 0,Y 531.129,Z 652.126,A -85,B 0,C 180,E1 -4317.725,E2 -4317.725} C_VEL
LIN {X 0,Y 531.147,Z 652.137,A -85,B 0,C 180,E1 -4320.758,E2 -4320.758} C_VEL
LIN {X 0,Y 531.1,Z 652.139,A -85,B 0,C 180,E1 -4323.034,E2 -4323.034} C_VEL
LIN {X 0,Y 531.082,Z 652.138,A -85,B 0,C 180,E1 -4326.077,E2 -4326.077} C_VEL
LIN {X 0,Y 531.028,Z 652.152,A -85,B 0,C 180,E1 -4329.138,E2 -4329.138} C_VEL
LIN {X 0,Y 531.051,Z 652.141,A -85,B 0,C 180,E1 -4331.678,E2 -4331.678} C_VEL
LIN {X 0,Y 531.019,Z 652.149,A -85,B 0,C 180,E1 -4334.956,E2 -4334.956} C_VEL
LIN {X 0,Y 531.006,Z 652.149,A -85,B 0,C 180,E1 -4337.723,E2 -4337.723} C_VEL
LIN {X 0,Y 530.992,Z 652.151,A -85,B 0,C 180,E1 -4340.938,E2 -4340.938} C_VEL
LIN {X 0,Y 530.97,Z 652.154,A -85,B 0,C 180,E1 -4344.225,E2 -4344.225} C_VEL
LIN {X 0,Y 531.002,Z 652.143,A -85,B 0,C 180,E1 -4346.744,E2 -4346.744} C_VEL
LIN {X 0,Y 530.991,Z 652.134,A -85,B 0,C 180,E1 -4349.322,E2 -4349.322} C_VEL
LIN {X 0,Y 530.972,Z 652.16,A -85,B 0,C 180,E1 -4352.104,E2 -4352.104} C_VEL
LIN {X 0,Y 530.983,Z 652.144,A -85,B 0,C 180,E1 -4354.855,E2 -4354.855} C_VEL
LIN {X 0,Y 530.96,Z 652.152,A -85,B 0,C 180,E1 -4357.508,E2 -4357.508} C_VEL
LIN {X 0,Y 531.021,Z 652.145,A -85,B 0,C 180,E1 -4360.429,E2 -4360.429} C_VEL
LIN {X 0,Y 530.961,Z 652.154,A -85,B 0,C 180,E1 -4363.495,E2 -4363.495} C_VEL
LIN {X 0,Y 530.96,Z 652.157,A -85,B 0,C 180,E1 -4366.506,E2 -4366.506} C_VEL
LIN {X 0,Y 530.983,Z 652.152,A -85,B 0,C 180,E1 -4368.976,E2 -4368.976} C_VEL
LIN {X 0,Y 530.954,Z 652.154,A -85,B 0,C 180,E1 -4371.53,E2 -4371.53} C_VEL
LIN {X 0,Y 530.977,Z 652.142,A -85,B 0,C 180,E1 -4374.383,E2 -4374.383} C_VEL
LIN {X 0,Y 530.996,Z 652.129,A -85,B 0,C 180,E1 -4377.552,E2 -4377.552} C_VEL
LIN {X 0,Y 531.02,Z 652.312,A -85,B 0,C 180,E1 -4377.89,E2 -4377.89} C_VEL
LIN {X 0,Y 532.691,Z 659.02,A -85,B 0,C 180,E1 -4379.045,E2 -4379.045} C_VEL
LIN {X 0,Y 534.387,Z 666.384,A -85,B 0,C 180,E1 -4380.227,E2 -4380.227} C_VEL
LIN {X 0,Y 533.873,Z 684.227,A -85,B 0,C 180,E1 -4382.778,E2 -4382.778} C_VEL
LIN {X 0,Y 533.562,Z 695.726,A -85,B 0,C 180,E1 -4384.378,E2 -4384.378} C_VEL
LIN {X 0,Y 534.469,Z 699.743,A -85,B 0,C 180,E1 -4384.515,E2 -4384.515} C_VEL
LIN {X 0,Y 537.359,Z 711.716,A -85,B 0,C 180,E1 -4384.834,E2 -4384.834} C_VEL
LIN {X 0,Y 536.008,Z 895.761,A -85,B 0,C 180,E1 -4387.423,E2 -4387.423} C_VEL
LIN {X 0,Y 535.728,Z 909.295,A -85,B 0,C 180,E1 -4387.691,E2 -4387.691} C_VEL
LIN {X 0,Y 535.455,Z 922.59,A -85,B 0,C 180,E1 -4388.059,E2 -4388.059} C_VEL
LIN {X 0,Y 535.047,Z 936.387,A -85,B 0,C 180,E1 -4388.552,E2 -4388.552} C_VEL
LIN {X 0,Y 534.619,Z 949.528,A -85,B 0,C 180,E1 -4389.137,E2 -4389.137} C_VEL
LIN {X 0,Y 534.156,Z 961.903,A -85,B 0,C 180,E1 -4389.796,E2 -4389.796} C_VEL
LIN {X 0,Y 533.693,Z 974.348,A -85,B 0,C 180,E1 -4390.58,E2 -4390.58} C_VEL
LIN {X 0,Y 533.253,Z 985.111,A -85,B 0,C 180,E1 -4391.362,E2 -4391.362} C_VEL
LIN {X 0,Y 532.842,Z 995.209,A -85,B 0,C 180,E1 -4392.197,E2 -4392.197} C_VEL
LIN {X 0,Y 532.357,Z 1005.055,A -85,B 0,C 180,E1 -4393.116,E2 -4393.116} C_VEL
LIN {X 0,Y 531.975,Z 1015.928,A -85,B 0,C 180,E1 -4394.287,E2 -4394.287} C_VEL
LIN {X 0,Y 531.613,Z 1025.386,A -85,B 0,C 180,E1 -4395.453,E2 -4395.453} C_VEL
LIN {X 0,Y 531.267,Z 1033.659,A -85,B 0,C 180,E1 -4396.615,E2 -4396.615} C_VEL
LIN {X 0,Y 531.077,Z 1040.913,A -85,B 0,C 180,E1 -4397.776,E2 -4397.776} C_VEL
LIN {X 0,Y 530.851,Z 1047.286,A -85,B 0,C 180,E1 -4398.933,E2 -4398.933} C_VEL
LIN {X 0,Y 530.653,Z 1054.459,A -85,B 0,C 180,E1 -4400.471,E2 -4400.471} C_VEL
LIN {X 0,Y 530.608,Z 1059.068,A -85,B 0,C 180,E1 -4401.623,E2 -4401.623} C_VEL
LIN {X 0,Y 530.546,Z 1064.086,A -85,B 0,C 180,E1 -4403.153,E2 -4403.153} C_VEL
LIN {X 0,Y 530.469,Z 1068.039,A -85,B 0,C 180,E1 -4404.679,E2 -4404.679} C_VEL
LIN {X 0,Y 530.478,Z 1070.942,A -85,B 0,C 180,E1 -4406.202,E2 -4406.202} C_VEL
LIN {X 0,Y 530.4,Z 1072.861,A -85,B 0,C 180,E1 -4407.722,E2 -4407.722} C_VEL
LIN {X 0,Y 530.341,Z 1073.814,A -85,B 0,C 180,E1 -4409.241,E2 -4409.241} C_VEL
LIN {X 0,Y 530.341,Z 1073.814,A -85,B 0,C 180,E1 -4410.759,E2 -4410.759} C_VEL
LIN {X 0,Y 530.4,Z 1072.861,A -85,B 0,C 180,E1 -4412.278,E2 -4412.278} C_VEL
LIN {X 0,Y 530.478,Z 1070.942,A -85,B 0,C 180,E1 -4413.798,E2 -4413.798} C_VEL
LIN {X 0,Y 530.469,Z 1068.039,A -85,B 0,C 180,E1 -4415.321,E2 -4415.321} C_VEL
LIN {X 0,Y 530.546,Z 1064.086,A -85,B 0,C 180,E1 -4416.847,E2 -4416.847} C_VEL
LIN {X 0,Y 530.608,Z 1059.068,A -85,B 0,C 180,E1 -4418.377,E2 -4418.377} C_VEL
LIN {X 0,Y 530.783,Z 1051.066,A -85,B 0,C 180,E1 -4420.297,E2 -4420.297} C_VEL
LIN {X 0,Y 531.012,Z 1043.087,A -85,B 0,C 180,E1 -4421.843,E2 -4421.843} C_VEL
LIN {X 0,Y 531.191,Z 1036.198,A -85,B 0,C 180,E1 -4422.998,E2 -4422.998} C_VEL
LIN {X 0,Y 531.53,Z 1026.841,A -85,B 0,C 180,E1 -4424.354,E2 -4424.354} C_VEL
LIN {X 0,Y 531.899,Z 1017.589,A -85,B 0,C 180,E1 -4425.519,E2 -4425.519} C_VEL
LIN {X 0,Y 532.238,Z 1008.846,A -85,B 0,C 180,E1 -4426.493,E2 -4426.493} C_VEL
LIN {X 0,Y 532.679,Z 997.861,A -85,B 0,C 180,E1 -4427.566,E2 -4427.566} C_VEL
LIN {X 0,Y 533.186,Z 986.352,A -85,B 0,C 180,E1 -4428.541,E2 -4428.541} C_VEL
LIN {X 0,Y 533.6,Z 975.781,A -85,B 0,C 180,E1 -4429.324,E2 -4429.324} C_VEL
LIN {X 0,Y 534.086,Z 963.574,A -85,B 0,C 180,E1 -4430.107,E2 -4430.107} C_VEL
LIN {X 0,Y 534.516,Z 952.953,A -85,B 0,C 180,E1 -4430.692,E2 -4430.692} C_VEL
LIN {X 0,Y 534.982,Z 939.413,A -85,B 0,C 180,E1 -4431.323,E2 -4431.323} C_VEL
LIN {X 0,Y 535.396,Z 926.315,A -85,B 0,C 180,E1 -4431.817,E2 -4431.817} C_VEL
LIN {X 0,Y 535.648,Z 913.207,A -85,B 0,C 180,E1 -4432.211,E2 -4432.211} C_VEL
LIN {X 0,Y 535.922,Z 899.976,A -85,B 0,C 180,E1 -4432.504,E2 -4432.504} C_VEL
LIN {X 0,Y 536.281,Z 866.371,A -85,B 0,C 180,E1 -4432.997,E2 -4432.997} C_VEL
LIN {X 0,Y 537.259,Z 710.823,A -85,B 0,C 180,E1 -4435.184,E2 -4435.184} C_VEL
LIN {X 0,Y 533.617,Z 696.048,A -85,B 0,C 180,E1 -4435.597,E2 -4435.597} C_VEL
LIN {X 0,Y 533.831,Z 685.708,A -85,B 0,C 180,E1 -4437.013,E2 -4437.013} C_VEL
LIN {X 0,Y 534.436,Z 667.373,A -85,B 0,C 180,E1 -4439.626,E2 -4439.626} C_VEL
LIN {X 0,Y 533.448,Z 661.949,A -85,B 0,C 180,E1 -4440.478,E2 -4440.478} C_VEL
LIN {X 0,Y 531.071,Z 652.614,A -85,B 0,C 180,E1 -4442.03,E2 -4442.03} C_VEL
LIN {X 0,Y 530.993,Z 652.14,A -85,B 0,C 180,E1 -4442.241,E2 -4442.241} C_VEL
LIN {X 0,Y 530.984,Z 652.155,A -85,B 0,C 180,E1 -4444.853,E2 -4444.853} C_VEL
LIN {X 0,Y 530.962,Z 652.145,A -85,B 0,C 180,E1 -4447.507,E2 -4447.507} C_VEL
LIN {X 0,Y 530.979,Z 652.151,A -85,B 0,C 180,E1 -4450.432,E2 -4450.432} C_VEL
LIN {X 0,Y 530.965,Z 652.161,A -85,B 0,C 180,E1 -4453.282,E2 -4453.282} C_VEL
LIN {X 0,Y 530.982,Z 652.156,A -85,B 0,C 180,E1 -4455.62,E2 -4455.62} C_VEL
LIN {X 0,Y 531.012,Z 652.139,A -85,B 0,C 180,E1 -4458.566,E2 -4458.566} C_VEL
LIN {X 0,Y 530.963,Z 652.156,A -85,B 0,C 180,E1 -4461.345,E2 -4461.345} C_VEL
LIN {X 0,Y 530.975,Z 652.147,A -85,B 0,C 180,E1 -4464.382,E2 -4464.382} C_VEL
LIN {X 0,Y 530.967,Z 652.153,A -85,B 0,C 180,E1 -4467.133,E2 -4467.133} C_VEL
LIN {X 0,Y 530.978,Z 652.152,A -85,B 0,C 180,E1 -4469.804,E2 -4469.804} C_VEL
LIN {X 0,Y 531.008,Z 652.145,A -85,B 0,C 180,E1 -4472.466,E2 -4472.466} C_VEL
LIN {X 0,Y 530.998,Z 652.15,A -85,B 0,C 180,E1 -4474.942,E2 -4474.942} C_VEL
LIN {X 0,Y 530.962,Z 652.155,A -85,B 0,C 180,E1 -4478.246,E2 -4478.246} C_VEL
LIN {X 0,Y 530.988,Z 652.155,A -85,B 0,C 180,E1 -4480.677,E2 -4480.677} C_VEL
LIN {X 0,Y 530.984,Z 652.154,A -85,B 0,C 180,E1 -4483.071,E2 -4483.071} C_VEL
LIN {X 0,Y 531.008,Z 652.147,A -85,B 0,C 180,E1 -4485.435,E2 -4485.435} C_VEL
LIN {X 0,Y 531.041,Z 652.145,A -85,B 0,C 180,E1 -4488.55,E2 -4488.55} C_VEL
LIN {X 0,Y 531.051,Z 652.137,A -85,B 0,C 180,E1 -4491.629,E2 -4491.629} C_VEL
LIN {X 0,Y 531.134,Z 652.134,A -85,B 0,C 180,E1 -4494.685,E2 -4494.685} C_VEL
LIN {X 0,Y 531.13,Z 652.133,A -85,B 0,C 180,E1 -4497.725,E2 -4497.725} C_VEL
LIN {X 0,Y 531.146,Z 652.131,A -85,B 0,C 180,E1 -4500.758,E2 -4500.758} C_VEL
LIN {X 0,Y 531.101,Z 652.133,A -85,B 0,C 180,E1 -4503.034,E2 -4503.034} C_VEL
LIN {X 0,Y 531.081,Z 652.139,A -85,B 0,C 180,E1 -4506.077,E2 -4506.077} C_VEL
LIN {X 0,Y 531.027,Z 652.144,A -85,B 0,C 180,E1 -4509.138,E2 -4509.138} C_VEL
LIN {X 0,Y 531.03,Z 652.143,A -85,B 0,C 180,E1 -4512.225,E2 -4512.225} C_VEL
LIN {X 0,Y 530.985,Z 652.151,A -85,B 0,C 180,E1 -4515.35,E2 -4515.35} C_VEL
LIN {X 0,Y 531.005,Z 652.149,A -85,B 0,C 180,E1 -4517.722,E2 -4517.722} C_VEL
LIN {X 0,Y 530.994,Z 652.148,A -85,B 0,C 180,E1 -4520.938,E2 -4520.938} C_VEL
LIN {X 0,Y 530.996,Z 652.153,A -85,B 0,C 180,E1 -4524.045,E2 -4524.045} C_VEL
LIN {X 0,Y 531.001,Z 652.144,A -85,B 0,C 180,E1 -4526.743,E2 -4526.743} C_VEL
LIN {X 0,Y 530.99,Z 652.139,A -85,B 0,C 180,E1 -4529.322,E2 -4529.322} C_VEL
LIN {X 0,Y 530.97,Z 652.154,A -85,B 0,C 180,E1 -4532.103,E2 -4532.103} C_VEL
LIN {X 0,Y 530.981,Z 652.148,A -85,B 0,C 180,E1 -4534.855,E2 -4534.855} C_VEL
LIN {X 0,Y 530.957,Z 652.152,A -85,B 0,C 180,E1 -4537.508,E2 -4537.508} C_VEL
LIN {X 0,Y 531,Z 652.151,A -85,B 0,C 180,E1 -4540.431,E2 -4540.431} C_VEL
LIN {X 0,Y 530.959,Z 652.158,A -85,B 0,C 180,E1 -4543.495,E2 -4543.495} C_VEL
LIN {X 0,Y 530.956,Z 652.158,A -85,B 0,C 180,E1 -4543.573,E2 -4543.573} C_VEL
LIN {X 0,Y 530.282,Z 652.24,A -85,B 0,C 180,E1 -4544.207,E2 -4544.207} C_VEL
LIN {X 0,Y 527.432,Z 652.602,A -85,B 0,C 180,E1 -4545.236,E2 -4545.236} C_VEL
LIN {X 0,Y 525.028,Z 652.9,A -85,B 0,C 180,E1 -4546.064,E2 -4546.064} C_VEL
LIN {X 0,Y 523.995,Z 653.026,A -85,B 0,C 180,E1 -4546.704,E2 -4546.704} C_VEL
LIN {X 0,Y 523.91,Z 653.036,A -85,B 0,C 180,E1 -4546.92,E2 -4546.92} C_VEL
LIN {X 0,Y 523.97,Z 653.027,A -85,B 0,C 180,E1 -4549.924,E2 -4549.924} C_VEL
LIN {X 0,Y 523.905,Z 653.035,A -85,B 0,C 180,E1 -4552.869,E2 -4552.869} C_VEL
LIN {X 0,Y 523.937,Z 653.037,A -85,B 0,C 180,E1 -4555.711,E2 -4555.711} C_VEL
LIN {X 0,Y 523.926,Z 653.031,A -85,B 0,C 180,E1 -4558.457,E2 -4558.457} C_VEL
LIN {X 0,Y 523.938,Z 653.03,A -85,B 0,C 180,E1 -4561.126,E2 -4561.126} C_VEL
LIN {X 0,Y 523.978,Z 653.031,A -85,B 0,C 180,E1 -4563.981,E2 -4563.981} C_VEL
LIN {X 0,Y 523.931,Z 653.036,A -85,B 0,C 180,E1 -4566.271,E2 -4566.271} C_VEL
LIN {X 0,Y 523.941,Z 653.03,A -85,B 0,C 180,E1 -4568.767,E2 -4568.767} C_VEL
LIN {X 0,Y 523.947,Z 653.029,A -85,B 0,C 180,E1 -4571.221,E2 -4571.221} C_VEL
LIN {X 0,Y 523.932,Z 653.031,A -85,B 0,C 180,E1 -4573.639,E2 -4573.639} C_VEL
LIN {X 0,Y 523.936,Z 653.034,A -85,B 0,C 180,E1 -4576.028,E2 -4576.028} C_VEL
LIN {X 0,Y 524.008,Z 653.028,A -85,B 0,C 180,E1 -4578.394,E2 -4578.394} C_VEL
LIN {X 0,Y 524.001,Z 653.022,A -85,B 0,C 180,E1 -4581.516,E2 -4581.516} C_VEL
LIN {X 0,Y 524.079,Z 653.018,A -85,B 0,C 180,E1 -4584.614,E2 -4584.614} C_VEL
LIN {X 0,Y 524.109,Z 653.009,A -85,B 0,C 180,E1 -4587.695,E2 -4587.695} C_VEL
LIN {X 0,Y 524.119,Z 653.013,A -85,B 0,C 180,E1 -4590.768,E2 -4590.768} C_VEL
LIN {X 0,Y 524.069,Z 653.02,A -85,B 0,C 180,E1 -4593.075,E2 -4593.075} C_VEL
LIN {X 0,Y 524.043,Z 653.017,A -85,B 0,C 180,E1 -4596.159,E2 -4596.159} C_VEL
LIN {X 0,Y 523.996,Z 653.029,A -85,B 0,C 180,E1 -4599.262,E2 -4599.262} C_VEL
LIN {X 0,Y 523.999,Z 653.028,A -85,B 0,C 180,E1 -4601.739,E2 -4601.739} C_VEL
LIN {X 0,Y 523.988,Z 653.026,A -85,B 0,C 180,E1 -4605.052,E2 -4605.052} C_VEL
LIN {X 0,Y 523.959,Z 653.033,A -85,B 0,C 180,E1 -4607.969,E2 -4607.969} C_VEL
LIN {X 0,Y 523.967,Z 653.028,A -85,B 0,C 180,E1 -4610.41,E2 -4610.41} C_VEL
LIN {X 0,Y 523.911,Z 653.033,A -85,B 0,C 180,E1 -4612.893,E2 -4612.893} C_VEL
LIN {X 0,Y 523.947,Z 653.03,A -85,B 0,C 180,E1 -4615.418,E2 -4615.418} C_VEL
LIN {X 0,Y 523.964,Z 653.033,A -85,B 0,C 180,E1 -4617.998,E2 -4617.998} C_VEL
LIN {X 0,Y 523.946,Z 653.03,A -85,B 0,C 180,E1 -4620.856,E2 -4620.856} C_VEL
LIN {X 0,Y 523.954,Z 653.029,A -85,B 0,C 180,E1 -4623.734,E2 -4623.734} C_VEL
LIN {X 0,Y 523.917,Z 653.04,A -85,B 0,C 180,E1 -4626.404,E2 -4626.404} C_VEL
LIN {X 0,Y 523.923,Z 653.033,A -85,B 0,C 180,E1 -4629.083,E2 -4629.083} C_VEL
LIN {X 0,Y 523.964,Z 653.027,A -85,B 0,C 180,E1 -4631.312,E2 -4631.312} C_VEL
LIN {X 0,Y 523.947,Z 653.036,A -85,B 0,C 180,E1 -4634.691,E2 -4634.691} C_VEL
LIN {X 0,Y 523.957,Z 653.027,A -85,B 0,C 180,E1 -4637.882,E2 -4637.882} C_VEL
LIN {X 0,Y 523.951,Z 653.035,A -85,B 0,C 180,E1 -4640.918,E2 -4640.918} C_VEL
LIN {X 0,Y 523.918,Z 653.019,A -85,B 0,C 180,E1 -4643.827,E2 -4643.827} C_VEL
LIN {X 0,Y 523.933,Z 653.029,A -85,B 0,C 180,E1 -4646.636,E2 -4646.636} C_VEL
LIN {X 0,Y 523.953,Z 653.026,A -85,B 0,C 180,E1 -4649.356,E2 -4649.356} C_VEL
LIN {X 0,Y 523.969,Z 653.015,A -85,B 0,C 180,E1 -4652.28,E2 -4652.28} C_VEL
LIN {X 0,Y 523.945,Z 653.027,A -85,B 0,C 180,E1 -4654.581,E2 -4654.581} C_VEL
LIN {X 0,Y 523.939,Z 653.028,A -85,B 0,C 180,E1 -4657.108,E2 -4657.108} C_VEL
LIN {X 0,Y 523.967,Z 653.033,A -85,B 0,C 180,E1 -4659.866,E2 -4659.866} C_VEL
LIN {X 0,Y 523.96,Z 653.022,A -85,B 0,C 180,E1 -4662.837,E2 -4662.837} C_VEL
LIN {X 0,Y 523.965,Z 653.024,A -85,B 0,C 180,E1 -4665.236,E2 -4665.236} C_VEL
LIN {X 0,Y 524,Z 653.026,A -85,B 0,C 180,E1 -4668.394,E2 -4668.394} C_VEL
LIN {X 0,Y 523.998,Z 653.018,A -85,B 0,C 180,E1 -4671.516,E2 -4671.516} C_VEL
LIN {X 0,Y 524.092,Z 653.015,A -85,B 0,C 180,E1 -4674.614,E2 -4674.614} C_VEL
LIN {X 0,Y 524.102,Z 653.001,A -85,B 0,C 180,E1 -4677.695,E2 -4677.695} C_VEL
LIN {X 0,Y 524.116,Z 653.012,A -85,B 0,C 180,E1 -4680.769,E2 -4680.769} C_VEL
LIN {X 0,Y 524.067,Z 653.014,A -85,B 0,C 180,E1 -4683.075,E2 -4683.075} C_VEL
LIN {X 0,Y 524.042,Z 653.015,A -85,B 0,C 180,E1 -4686.159,E2 -4686.159} C_VEL
LIN {X 0,Y 523.995,Z 653.026,A -85,B 0,C 180,E1 -4689.262,E2 -4689.262} C_VEL
LIN {X 0,Y 524.013,Z 653.016,A -85,B 0,C 180,E1 -4691.752,E2 -4691.752} C_VEL
LIN {X 0,Y 523.981,Z 653.027,A -85,B 0,C 180,E1 -4695.053,E2 -4695.053} C_VEL
LIN {X 0,Y 523.954,Z 653.024,A -85,B 0,C 180,E1 -4697.969,E2 -4697.969} C_VEL
LIN {X 0,Y 523.962,Z 653.025,A -85,B 0,C 180,E1 -4700.41,E2 -4700.41} C_VEL
LIN {X 0,Y 523.907,Z 653.028,A -85,B 0,C 180,E1 -4702.894,E2 -4702.894} C_VEL
LIN {X 0,Y 523.946,Z 653.033,A -85,B 0,C 180,E1 -4705.419,E2 -4705.419} C_VEL
LIN {X 0,Y 523.962,Z 653.012,A -85,B 0,C 180,E1 -4707.999,E2 -4707.999} C_VEL
LIN {X 0,Y 523.944,Z 653.024,A -85,B 0,C 180,E1 -4710.857,E2 -4710.857} C_VEL
LIN {X 0,Y 523.955,Z 653.032,A -85,B 0,C 180,E1 -4713.736,E2 -4713.736} C_VEL
LIN {X 0,Y 523.917,Z 653.03,A -85,B 0,C 180,E1 -4716.405,E2 -4716.405} C_VEL
LIN {X 0,Y 523.953,Z 653.027,A -85,B 0,C 180,E1 -4719.082,E2 -4719.082} C_VEL
LIN {X 0,Y 523.96,Z 653.024,A -85,B 0,C 180,E1 -4722.118,E2 -4722.118} C_VEL
LIN {X 0,Y 523.949,Z 653.02,A -85,B 0,C 180,E1 -4725.309,E2 -4725.309} C_VEL
LIN {X 0,Y 523.956,Z 653.028,A -85,B 0,C 180,E1 -4728.69,E2 -4728.69} C_VEL
LIN {X 0,Y 523.912,Z 653.031,A -85,B 0,C 180,E1 -4731.899,E2 -4731.899} C_VEL
LIN {X 0,Y 523.934,Z 653.027,A -85,B 0,C 180,E1 -4734.91,E2 -4734.91} C_VEL
LIN {X 0,Y 523.967,Z 653.126,A -85,B 0,C 180,E1 -4737.554,E2 -4737.554} C_VEL
LIN {X 0,Y 524.605,Z 655.743,A -85,B 0,C 180,E1 -4738.051,E2 -4738.051} C_VEL
LIN {X 0,Y 527.471,Z 667.558,A -85,B 0,C 180,E1 -4740.003,E2 -4740.003} C_VEL
LIN {X 0,Y 527.412,Z 675.122,A -85,B 0,C 180,E1 -4741.116,E2 -4741.116} C_VEL
LIN {X 0,Y 526.737,Z 695.441,A -85,B 0,C 180,E1 -4744.019,E2 -4744.019} C_VEL
LIN {X 0,Y 527.619,Z 699.43,A -85,B 0,C 180,E1 -4744.158,E2 -4744.158} C_VEL
LIN {X 0,Y 530.823,Z 712.274,A -85,B 0,C 180,E1 -4744.513,E2 -4744.513} C_VEL
LIN {X 0,Y 529.732,Z 869.948,A -85,B 0,C 180,E1 -4746.754,E2 -4746.754} C_VEL
LIN {X 0,Y 529.385,Z 899.936,A -85,B 0,C 180,E1 -4747.202,E2 -4747.202} C_VEL
LIN {X 0,Y 529.087,Z 913.177,A -85,B 0,C 180,E1 -4747.498,E2 -4747.498} C_VEL
LIN {X 0,Y 528.765,Z 926.298,A -85,B 0,C 180,E1 -4747.895,E2 -4747.895} C_VEL
LIN {X 0,Y 528.345,Z 938.687,A -85,B 0,C 180,E1 -4748.366,E2 -4748.366} C_VEL
LIN {X 0,Y 527.908,Z 950.968,A -85,B 0,C 180,E1 -4748.934,E2 -4748.934} C_VEL
LIN {X 0,Y 527.445,Z 961.889,A -85,B 0,C 180,E1 -4749.527,E2 -4749.527} C_VEL
LIN {X 0,Y 526.995,Z 972.906,A -85,B 0,C 180,E1 -4750.221,E2 -4750.221} C_VEL
LIN {X 0,Y 526.506,Z 983.859,A -85,B 0,C 180,E1 -4751.013,E2 -4751.013} C_VEL
LIN {X 0,Y 525.98,Z 995.364,A -85,B 0,C 180,E1 -4751.972,E2 -4751.972} C_VEL
LIN {X 0,Y 525.479,Z 1005.047,A -85,B 0,C 180,E1 -4752.889,E2 -4752.889} C_VEL
LIN {X 0,Y 525.047,Z 1015.92,A -85,B 0,C 180,E1 -4754.074,E2 -4754.074} C_VEL
LIN {X 0,Y 524.741,Z 1023.639,A -85,B 0,C 180,E1 -4755.021,E2 -4755.021} C_VEL
LIN {X 0,Y 524.336,Z 1032.383,A -85,B 0,C 180,E1 -4756.237,E2 -4756.237} C_VEL
LIN {X 0,Y 524.03,Z 1040.907,A -85,B 0,C 180,E1 -4757.609,E2 -4757.609} C_VEL
LIN {X 0,Y 523.821,Z 1047.28,A -85,B 0,C 180,E1 -4758.782,E2 -4758.782} C_VEL
LIN {X 0,Y 523.595,Z 1054.455,A -85,B 0,C 180,E1 -4760.341,E2 -4760.341} C_VEL
LIN {X 0,Y 523.529,Z 1059.062,A -85,B 0,C 180,E1 -4761.508,E2 -4761.508} C_VEL
LIN {X 0,Y 523.477,Z 1064.082,A -85,B 0,C 180,E1 -4763.06,E2 -4763.06} C_VEL
LIN {X 0,Y 523.397,Z 1068.033,A -85,B 0,C 180,E1 -4764.607,E2 -4764.607} C_VEL
LIN {X 0,Y 523.399,Z 1070.938,A -85,B 0,C 180,E1 -4766.15,E2 -4766.15} C_VEL
LIN {X 0,Y 523.324,Z 1072.857,A -85,B 0,C 180,E1 -4767.691,E2 -4767.691} C_VEL
LIN {X 0,Y 523.247,Z 1073.809,A -85,B 0,C 180,E1 -4769.23,E2 -4769.23} C_VEL
LIN {X 0,Y 523.247,Z 1073.809,A -85,B 0,C 180,E1 -4770.77,E2 -4770.77} C_VEL
LIN {X 0,Y 523.324,Z 1072.857,A -85,B 0,C 180,E1 -4772.309,E2 -4772.309} C_VEL
LIN {X 0,Y 523.399,Z 1070.938,A -85,B 0,C 180,E1 -4773.85,E2 -4773.85} C_VEL
LIN {X 0,Y 523.397,Z 1068.033,A -85,B 0,C 180,E1 -4775.393,E2 -4775.393} C_VEL
LIN {X 0,Y 523.477,Z 1064.082,A -85,B 0,C 180,E1 -4776.94,E2 -4776.94} C_VEL
LIN {X 0,Y 523.529,Z 1059.062,A -85,B 0,C 180,E1 -4778.492,E2 -4778.492} C_VEL
LIN {X 0,Y 523.725,Z 1051.065,A -85,B 0,C 180,E1 -4780.437,E2 -4780.437} C_VEL
LIN {X 0,Y 523.995,Z 1043.112,A -85,B 0,C 180,E1 -4781.998,E2 -4781.998} C_VEL
LIN {X 0,Y 524.171,Z 1036.191,A -85,B 0,C 180,E1 -4783.175,E2 -4783.175} C_VEL
LIN {X 0,Y 524.518,Z 1028.289,A -85,B 0,C 180,E1 -4784.352,E2 -4784.352} C_VEL
LIN {X 0,Y 524.891,Z 1019.243,A -85,B 0,C 180,E1 -4785.532,E2 -4785.532} C_VEL
LIN {X 0,Y 525.345,Z 1008.837,A -85,B 0,C 180,E1 -4786.715,E2 -4786.715} C_VEL
LIN {X 0,Y 525.773,Z 998.935,A -85,B 0,C 180,E1 -4787.703,E2 -4787.703} C_VEL
LIN {X 0,Y 526.346,Z 987.583,A -85,B 0,C 180,E1 -4788.69,E2 -4788.69} C_VEL
LIN {X 0,Y 526.856,Z 975.771,A -85,B 0,C 180,E1 -4789.581,E2 -4789.581} C_VEL
LIN {X 0,Y 527.361,Z 963.56,A -85,B 0,C 180,E1 -4790.374,E2 -4790.374} C_VEL
LIN {X 0,Y 527.846,Z 952.944,A -85,B 0,C 180,E1 -4790.966,E2 -4790.966} C_VEL
LIN {X 0,Y 528.328,Z 939.727,A -85,B 0,C 180,E1 -4791.59,E2 -4791.59} C_VEL
LIN {X 0,Y 528.777,Z 927.043,A -85,B 0,C 180,E1 -4792.079,E2 -4792.079} C_VEL
LIN {X 0,Y 529.075,Z 913.177,A -85,B 0,C 180,E1 -4792.502,E2 -4792.502} C_VEL
LIN {X 0,Y 529.38,Z 899.936,A -85,B 0,C 180,E1 -4792.798,E2 -4792.798} C_VEL
LIN {X 0,Y 529.723,Z 868.159,A -85,B 0,C 180,E1 -4793.273,E2 -4793.273} C_VEL
LIN {X 0,Y 530.883,Z 712.314,A -85,B 0,C 180,E1 -4795.484,E2 -4795.484} C_VEL
LIN {X 0,Y 526.76,Z 695.639,A -85,B 0,C 180,E1 -4795.964,E2 -4795.964} C_VEL
LIN {X 0,Y 527.453,Z 675.123,A -85,B 0,C 180,E1 -4798.881,E2 -4798.881} C_VEL
LIN {X 0,Y 527.495,Z 667.518,A -85,B 0,C 180,E1 -4800.001,E2 -4800.001} C_VEL
LIN {X 0,Y 524.041,Z 653.511,A -85,B 0,C 180,E1 -4802.339,E2 -4802.339} C_VEL
LIN {X 0,Y 523.941,Z 653.015,A -85,B 0,C 180,E1 -4802.562,E2 -4802.562} C_VEL
LIN {X 0,Y 523.931,Z 653.024,A -85,B 0,C 180,E1 -4805.225,E2 -4805.225} C_VEL
LIN {X 0,Y 523.912,Z 653.031,A -85,B 0,C 180,E1 -4808.101,E2 -4808.101} C_VEL
LIN {X 0,Y 523.956,Z 653.028,A -85,B 0,C 180,E1 -4811.31,E2 -4811.31} C_VEL
LIN {X 0,Y 523.949,Z 653.019,A -85,B 0,C 180,E1 -4814.691,E2 -4814.691} C_VEL
LIN {X 0,Y 523.96,Z 653.024,A -85,B 0,C 180,E1 -4817.882,E2 -4817.882} C_VEL
LIN {X 0,Y 523.953,Z 653.027,A -85,B 0,C 180,E1 -4820.918,E2 -4820.918} C_VEL
LIN {X 0,Y 523.922,Z 653.027,A -85,B 0,C 180,E1 -4823.827,E2 -4823.827} C_VEL
LIN {X 0,Y 523.936,Z 653.03,A -85,B 0,C 180,E1 -4826.635,E2 -4826.635} C_VEL
LIN {X 0,Y 523.955,Z 653.023,A -85,B 0,C 180,E1 -4829.356,E2 -4829.356} C_VEL
LIN {X 0,Y 523.971,Z 653.016,A -85,B 0,C 180,E1 -4832.28,E2 -4832.28} C_VEL
LIN {X 0,Y 523.946,Z 653.033,A -85,B 0,C 180,E1 -4834.581,E2 -4834.581} C_VEL
LIN {X 0,Y 523.907,Z 653.028,A -85,B 0,C 180,E1 -4837.106,E2 -4837.106} C_VEL
LIN {X 0,Y 523.969,Z 653.025,A -85,B 0,C 180,E1 -4839.865,E2 -4839.865} C_VEL
LIN {X 0,Y 523.961,Z 653.031,A -85,B 0,C 180,E1 -4842.837,E2 -4842.837} C_VEL
LIN {X 0,Y 523.966,Z 653.026,A -85,B 0,C 180,E1 -4845.235,E2 -4845.235} C_VEL
LIN {X 0,Y 524.002,Z 653.02,A -85,B 0,C 180,E1 -4848.394,E2 -4848.394} C_VEL
LIN {X 0,Y 523.998,Z 653.016,A -85,B 0,C 180,E1 -4851.516,E2 -4851.516} C_VEL
LIN {X 0,Y 524.093,Z 653.01,A -85,B 0,C 180,E1 -4854.614,E2 -4854.614} C_VEL
LIN {X 0,Y 524.102,Z 653.008,A -85,B 0,C 180,E1 -4857.694,E2 -4857.694} C_VEL
LIN {X 0,Y 524.116,Z 653.007,A -85,B 0,C 180,E1 -4860.768,E2 -4860.768} C_VEL
LIN {X 0,Y 524.067,Z 653.009,A -85,B 0,C 180,E1 -4863.075,E2 -4863.075} C_VEL
LIN {X 0,Y 524.042,Z 653.015,A -85,B 0,C 180,E1 -4866.159,E2 -4866.159} C_VEL
LIN {X 0,Y 523.994,Z 653.021,A -85,B 0,C 180,E1 -4869.262,E2 -4869.262} C_VEL
LIN {X 0,Y 523.996,Z 653.026,A -85,B 0,C 180,E1 -4871.743,E2 -4871.743} C_VEL
LIN {X 0,Y 523.98,Z 653.022,A -85,B 0,C 180,E1 -4875.052,E2 -4875.052} C_VEL
LIN {X 0,Y 523.953,Z 653.029,A -85,B 0,C 180,E1 -4877.969,E2 -4877.969} C_VEL
LIN {X 0,Y 523.962,Z 653.03,A -85,B 0,C 180,E1 -4880.41,E2 -4880.41} C_VEL
LIN {X 0,Y 523.939,Z 653.028,A -85,B 0,C 180,E1 -4882.892,E2 -4882.892} C_VEL
LIN {X 0,Y 523.975,Z 653.027,A -85,B 0,C 180,E1 -4886.021,E2 -4886.021} C_VEL
LIN {X 0,Y 523.94,Z 653.017,A -85,B 0,C 180,E1 -4888.874,E2 -4888.874} C_VEL
LIN {X 0,Y 523.922,Z 653.03,A -85,B 0,C 180,E1 -4891.544,E2 -4891.544} C_VEL
LIN {X 0,Y 523.936,Z 653.03,A -85,B 0,C 180,E1 -4894.289,E2 -4894.289} C_VEL
LIN {X 0,Y 523.902,Z 653.031,A -85,B 0,C 180,E1 -4897.132,E2 -4897.132} C_VEL
LIN {X 0,Y 523.958,Z 653.026,A -85,B 0,C 180,E1 -4900.134,E2 -4900.134} C_VEL
LIN {X 0,Y 523.936,Z 653.031,A -85,B 0,C 180,E1 -4902.461,E2 -4902.461} C_VEL
LIN {X 0,Y 523.947,Z 653.036,A -85,B 0,C 180,E1 -4905.309,E2 -4905.309} C_VEL
LIN {X 0,Y 523.91,Z 653.036,A -85,B 0,C 180,E1 -4906.92,E2 -4906.92} C_VEL
LIN {X 0,Y 523.249,Z 653.12,A -85,B 0,C 180,E1 -4907.562,E2 -4907.562} C_VEL
LIN {X 0,Y 520.421,Z 653.469,A -85,B 0,C 180,E1 -4908.604,E2 -4908.604} C_VEL
LIN {X 0,Y 518.023,Z 653.773,A -85,B 0,C 180,E1 -4909.443,E2 -4909.443} C_VEL
LIN {X 0,Y 516.984,Z 653.897,A -85,B 0,C 180,E1 -4910.091,E2 -4910.091} C_VEL
LIN {X 0,Y 516.893,Z 653.906,A -85,B 0,C 180,E1 -4910.31,E2 -4910.31} C_VEL
LIN {X 0,Y 516.878,Z 653.915,A -85,B 0,C 180,E1 -4913.342,E2 -4913.342} C_VEL
LIN {X 0,Y 516.905,Z 653.909,A -85,B 0,C 180,E1 -4916.122,E2 -4916.122} C_VEL
LIN {X 0,Y 516.888,Z 653.908,A -85,B 0,C 180,E1 -4918.935,E2 -4918.935} C_VEL
LIN {X 0,Y 516.915,Z 653.91,A -85,B 0,C 180,E1 -4921.585,E2 -4921.585} C_VEL
LIN {X 0,Y 516.926,Z 653.909,A -85,B 0,C 180,E1 -4924.211,E2 -4924.211} C_VEL
LIN {X 0,Y 516.867,Z 653.912,A -85,B 0,C 180,E1 -4926.777,E2 -4926.777} C_VEL
LIN {X 0,Y 516.934,Z 653.905,A -85,B 0,C 180,E1 -4929.732,E2 -4929.732} C_VEL
LIN {X 0,Y 516.924,Z 653.908,A -85,B 0,C 180,E1 -4932.596,E2 -4932.596} C_VEL
LIN {X 0,Y 516.938,Z 653.904,A -85,B 0,C 180,E1 -4935.03,E2 -4935.03} C_VEL
LIN {X 0,Y 516.961,Z 653.904,A -85,B 0,C 180,E1 -4938.234,E2 -4938.234} C_VEL
LIN {X 0,Y 516.966,Z 653.899,A -85,B 0,C 180,E1 -4941.4,E2 -4941.4} C_VEL
LIN {X 0,Y 517.007,Z 653.893,A -85,B 0,C 180,E1 -4943.757,E2 -4943.757} C_VEL
LIN {X 0,Y 517.081,Z 653.884,A -85,B 0,C 180,E1 -4947.663,E2 -4947.663} C_VEL
LIN {X 0,Y 517.089,Z 653.889,A -85,B 0,C 180,E1 -4950.779,E2 -4950.779} C_VEL
LIN {X 0,Y 517.01,Z 653.899,A -85,B 0,C 180,E1 -4953.117,E2 -4953.117} C_VEL
LIN {X 0,Y 517.007,Z 653.893,A -85,B 0,C 180,E1 -4956.243,E2 -4956.243} C_VEL
LIN {X 0,Y 516.95,Z 653.908,A -85,B 0,C 180,E1 -4959.389,E2 -4959.389} C_VEL
LIN {X 0,Y 516.948,Z 653.905,A -85,B 0,C 180,E1 -4961.807,E2 -4961.807} C_VEL
LIN {X 0,Y 516.94,Z 653.905,A -85,B 0,C 180,E1 -4965.146,E2 -4965.146} C_VEL
LIN {X 0,Y 516.92,Z 653.907,A -85,B 0,C 180,E1 -4968.222,E2 -4968.222} C_VEL
LIN {X 0,Y 516.907,Z 653.906,A -85,B 0,C 180,E1 -4970.701,E2 -4970.701} C_VEL
LIN {X 0,Y 516.906,Z 653.913,A -85,B 0,C 180,E1 -4974.072,E2 -4974.072} C_VEL
LIN {X 0,Y 516.921,Z 653.906,A -85,B 0,C 180,E1 -4976.657,E2 -4976.657} C_VEL
LIN {X 0,Y 516.919,Z 653.905,A -85,B 0,C 180,E1 -4979.526,E2 -4979.526} C_VEL
LIN {X 0,Y 516.894,Z 653.913,A -85,B 0,C 180,E1 -4982.544,E2 -4982.544} C_VEL
LIN {X 0,Y 516.876,Z 653.909,A -85,B 0,C 180,E1 -4985.332,E2 -4985.332} C_VEL
LIN {X 0,Y 516.874,Z 653.911,A -85,B 0,C 180,E1 -4987.943,E2 -4987.943} C_VEL
LIN {X 0,Y 516.896,Z 653.914,A -85,B 0,C 180,E1 -4990.739,E2 -4990.739} C_VEL
LIN {X 0,Y 516.874,Z 653.909,A -85,B 0,C 180,E1 -4993.903,E2 -4993.903} C_VEL
LIN {X 0,Y 516.874,Z 653.91,A -85,B 0,C 180,E1 -4996.106,E2 -4996.106} C_VEL
LIN {X 0,Y 516.899,Z 653.911,A -85,B 0,C 180,E1 -4999.26,E2 -4999.26} C_VEL
LIN {X 0,Y 516.872,Z 653.905,A -85,B 0,C 180,E1 -5002.056,E2 -5002.056} C_VEL
LIN {X 0,Y 516.886,Z 653.902,A -85,B 0,C 180,E1 -5005.176,E2 -5005.176} C_VEL
LIN {X 0,Y 516.872,Z 653.909,A -85,B 0,C 180,E1 -5007.975,E2 -5007.975} C_VEL
LIN {X 0,Y 516.925,Z 653.89,A -85,B 0,C 180,E1 -5010.696,E2 -5010.696} C_VEL
LIN {X 0,Y 516.934,Z 653.906,A -85,B 0,C 180,E1 -5013.803,E2 -5013.803} C_VEL
LIN {X 0,Y 516.884,Z 653.905,A -85,B 0,C 180,E1 -5016.778,E2 -5016.778} C_VEL
LIN {X 0,Y 516.928,Z 653.909,A -85,B 0,C 180,E1 -5019.731,E2 -5019.731} C_VEL
LIN {X 0,Y 516.92,Z 653.899,A -85,B 0,C 180,E1 -5022.596,E2 -5022.596} C_VEL
LIN {X 0,Y 516.93,Z 653.9,A -85,B 0,C 180,E1 -5025.03,E2 -5025.03} C_VEL
LIN {X 0,Y 516.953,Z 653.902,A -85,B 0,C 180,E1 -5028.234,E2 -5028.234} C_VEL
LIN {X 0,Y 516.962,Z 653.893,A -85,B 0,C 180,E1 -5031.4,E2 -5031.4} C_VEL
LIN {X 0,Y 517.053,Z 653.893,A -85,B 0,C 180,E1 -5034.54,E2 -5034.54} C_VEL
LIN {X 0,Y 517.074,Z 653.876,A -85,B 0,C 180,E1 -5037.663,E2 -5037.663} C_VEL
LIN {X 0,Y 517.086,Z 653.888,A -85,B 0,C 180,E1 -5040.779,E2 -5040.779} C_VEL
LIN {X 0,Y 517.007,Z 653.893,A -85,B 0,C 180,E1 -5043.117,E2 -5043.117} C_VEL
LIN {X 0,Y 517.005,Z 653.892,A -85,B 0,C 180,E1 -5046.243,E2 -5046.243} C_VEL
LIN {X 0,Y 516.95,Z 653.902,A -85,B 0,C 180,E1 -5049.389,E2 -5049.389} C_VEL
LIN {X 0,Y 516.972,Z 653.893,A -85,B 0,C 180,E1 -5051.824,E2 -5051.824} C_VEL
LIN {X 0,Y 516.933,Z 653.907,A -85,B 0,C 180,E1 -5055.147,E2 -5055.147} C_VEL
LIN {X 0,Y 516.916,Z 653.899,A -85,B 0,C 180,E1 -5058.223,E2 -5058.223} C_VEL
LIN {X 0,Y 516.903,Z 653.905,A -85,B 0,C 180,E1 -5060.702,E2 -5060.702} C_VEL
LIN {X 0,Y 516.901,Z 653.908,A -85,B 0,C 180,E1 -5064.073,E2 -5064.073} C_VEL
LIN {X 0,Y 516.92,Z 653.897,A -85,B 0,C 180,E1 -5066.658,E2 -5066.658} C_VEL
LIN {X 0,Y 516.916,Z 653.887,A -85,B 0,C 180,E1 -5069.527,E2 -5069.527} C_VEL
LIN {X 0,Y 516.893,Z 653.908,A -85,B 0,C 180,E1 -5072.545,E2 -5072.545} C_VEL
LIN {X 0,Y 516.876,Z 653.9,A -85,B 0,C 180,E1 -5075.333,E2 -5075.333} C_VEL
LIN {X 0,Y 516.875,Z 653.911,A -85,B 0,C 180,E1 -5077.944,E2 -5077.944} C_VEL
LIN {X 0,Y 516.91,Z 653.897,A -85,B 0,C 180,E1 -5080.739,E2 -5080.739} C_VEL
LIN {X 0,Y 516.877,Z 653.912,A -85,B 0,C 180,E1 -5083.904,E2 -5083.904} C_VEL
LIN {X 0,Y 516.876,Z 653.904,A -85,B 0,C 180,E1 -5086.108,E2 -5086.108} C_VEL
LIN {X 0,Y 516.912,Z 653.908,A -85,B 0,C 180,E1 -5088.399,E2 -5088.399} C_VEL
LIN {X 0,Y 516.877,Z 653.909,A -85,B 0,C 180,E1 -5091.285,E2 -5091.285} C_VEL
LIN {X 0,Y 516.886,Z 653.89,A -85,B 0,C 180,E1 -5094.222,E2 -5094.222} C_VEL
LIN {X 0,Y 516.922,Z 654.003,A -85,B 0,C 180,E1 -5097.232,E2 -5097.232} C_VEL
LIN {X 0,Y 518.039,Z 658.495,A -85,B 0,C 180,E1 -5098.057,E2 -5098.057} C_VEL
LIN {X 0,Y 520.853,Z 670.457,A -85,B 0,C 180,E1 -5100.05,E2 -5100.05} C_VEL
LIN {X 0,Y 520.201,Z 688.247,A -85,B 0,C 180,E1 -5102.656,E2 -5102.656} C_VEL
LIN {X 0,Y 520.008,Z 695.456,A -85,B 0,C 180,E1 -5103.676,E2 -5103.676} C_VEL
LIN {X 0,Y 524.408,Z 713.566,A -85,B 0,C 180,E1 -5104.2,E2 -5104.2} C_VEL
LIN {X 0,Y 523.078,Z 885.939,A -85,B 0,C 180,E1 -5106.676,E2 -5106.676} C_VEL
LIN {X 0,Y 522.668,Z 907.212,A -85,B 0,C 180,E1 -5107.05,E2 -5107.05} C_VEL
LIN {X 0,Y 522.307,Z 921.77,A -85,B 0,C 180,E1 -5107.451,E2 -5107.451} C_VEL
LIN {X 0,Y 521.834,Z 935.537,A -85,B 0,C 180,E1 -5107.946,E2 -5107.946} C_VEL
LIN {X 0,Y 521.382,Z 947.966,A -85,B 0,C 180,E1 -5108.501,E2 -5108.501} C_VEL
LIN {X 0,Y 520.844,Z 960.205,A -85,B 0,C 180,E1 -5109.153,E2 -5109.153} C_VEL
LIN {X 0,Y 520.277,Z 972.896,A -85,B 0,C 180,E1 -5109.955,E2 -5109.955} C_VEL
LIN {X 0,Y 519.715,Z 983.848,A -85,B 0,C 180,E1 -5110.755,E2 -5110.755} C_VEL
LIN {X 0,Y 519.201,Z 994.293,A -85,B 0,C 180,E1 -5111.628,E2 -5111.628} C_VEL
LIN {X 0,Y 518.628,Z 1005.039,A -85,B 0,C 180,E1 -5112.655,E2 -5112.655} C_VEL
LIN {X 0,Y 518.149,Z 1015.913,A -85,B 0,C 180,E1 -5113.856,E2 -5113.856} C_VEL
LIN {X 0,Y 517.77,Z 1023.916,A -85,B 0,C 180,E1 -5114.853,E2 -5114.853} C_VEL
LIN {X 0,Y 517.331,Z 1032.376,A -85,B 0,C 180,E1 -5116.047,E2 -5116.047} C_VEL
LIN {X 0,Y 516.992,Z 1040.902,A -85,B 0,C 180,E1 -5117.438,E2 -5117.438} C_VEL
LIN {X 0,Y 516.801,Z 1047.274,A -85,B 0,C 180,E1 -5118.628,E2 -5118.628} C_VEL
LIN {X 0,Y 516.552,Z 1054.451,A -85,B 0,C 180,E1 -5120.208,E2 -5120.208} C_VEL
LIN {X 0,Y 516.465,Z 1059.056,A -85,B 0,C 180,E1 -5121.391,E2 -5121.391} C_VEL
LIN {X 0,Y 516.386,Z 1064.078,A -85,B 0,C 180,E1 -5122.964,E2 -5122.964} C_VEL
LIN {X 0,Y 516.304,Z 1068.028,A -85,B 0,C 180,E1 -5124.532,E2 -5124.532} C_VEL
LIN {X 0,Y 516.304,Z 1070.933,A -85,B 0,C 180,E1 -5126.097,E2 -5126.097} C_VEL
LIN {X 0,Y 516.251,Z 1072.852,A -85,B 0,C 180,E1 -5127.659,E2 -5127.659} C_VEL
LIN {X 0,Y 516.157,Z 1073.804,A -85,B 0,C 180,E1 -5129.22,E2 -5129.22} C_VEL
LIN {X 0,Y 516.149,Z 1074,A -85,B 0,C 180,E1 -5130,E2 -5130} C_VEL
LIN {X 0,Y 516.186,Z 1073.513,A -85,B 0,C 180,E1 -5131.56,E2 -5131.56} C_VEL
LIN {X 0,Y 516.268,Z 1072.082,A -85,B 0,C 180,E1 -5133.121,E2 -5133.121} C_VEL
LIN {X 0,Y 516.226,Z 1069.668,A -85,B 0,C 180,E1 -5134.685,E2 -5134.685} C_VEL
LIN {X 0,Y 516.368,Z 1065.524,A -85,B 0,C 180,E1 -5136.507,E2 -5136.507} C_VEL
LIN {X 0,Y 516.41,Z 1061.719,A -85,B 0,C 180,E1 -5137.822,E2 -5137.822} C_VEL
LIN {X 0,Y 516.49,Z 1056.055,A -85,B 0,C 180,E1 -5139.397,E2 -5139.397} C_VEL
LIN {X 0,Y 516.675,Z 1051.058,A -85,B 0,C 180,E1 -5140.581,E2 -5140.581} C_VEL
LIN {X 0,Y 516.976,Z 1043.104,A -85,B 0,C 180,E1 -5142.164,E2 -5142.164} C_VEL
LIN {X 0,Y 517.19,Z 1036.185,A -85,B 0,C 180,E1 -5143.356,E2 -5143.356} C_VEL
LIN {X 0,Y 517.542,Z 1028.281,A -85,B 0,C 180,E1 -5144.549,E2 -5144.549} C_VEL
LIN {X 0,Y 517.971,Z 1019.235,A -85,B 0,C 180,E1 -5145.745,E2 -5145.745} C_VEL
LIN {X 0,Y 518.45,Z 1008.829,A -85,B 0,C 180,E1 -5146.944,E2 -5146.944} C_VEL
LIN {X 0,Y 518.942,Z 998.926,A -85,B 0,C 180,E1 -5147.944,E2 -5147.944} C_VEL
LIN {X 0,Y 519.554,Z 987.572,A -85,B 0,C 180,E1 -5148.944,E2 -5148.944} C_VEL
LIN {X 0,Y 520.036,Z 977.194,A -85,B 0,C 180,E1 -5149.746,E2 -5149.746} C_VEL
LIN {X 0,Y 520.601,Z 965.216,A -85,B 0,C 180,E1 -5150.548,E2 -5150.548} C_VEL
LIN {X 0,Y 521.181,Z 952.934,A -85,B 0,C 180,E1 -5151.247,E2 -5151.247} C_VEL
LIN {X 0,Y 521.702,Z 940.076,A -85,B 0,C 180,E1 -5151.862,E2 -5151.862} C_VEL
LIN {X 0,Y 522.175,Z 926.997,A -85,B 0,C 180,E1 -5152.373,E2 -5152.373} C_VEL
LIN {X 0,Y 522.497,Z 914.07,A -85,B 0,C 180,E1 -5152.775,E2 -5152.775} C_VEL
LIN {X 0,Y 522.811,Z 901.231,A -85,B 0,C 180,E1 -5153.075,E2 -5153.075} C_VEL
LIN {X 0,Y 523.207,Z 875.195,A -85,B 0,C 180,E1 -5153.475,E2 -5153.475} C_VEL
LIN {X 0,Y 524.414,Z 713.456,A -85,B 0,C 180,E1 -5155.801,E2 -5155.801} C_VEL
LIN {X 0,Y 519.964,Z 695.307,A -85,B 0,C 180,E1 -5156.335,E2 -5156.335} C_VEL
LIN {X 0,Y 520.742,Z 674.909,A -85,B 0,C 180,E1 -5159.289,E2 -5159.289} C_VEL
LIN {X 0,Y 520.884,Z 670.458,A -85,B 0,C 180,E1 -5159.948,E2 -5159.948} C_VEL
LIN {X 0,Y 518.293,Z 659.562,A -85,B 0,C 180,E1 -5161.766,E2 -5161.766} C_VEL
LIN {X 0,Y 516.984,Z 654.22,A -85,B 0,C 180,E1 -5162.705,E2 -5162.705} C_VEL
LIN {X 0,Y 516.91,Z 653.883,A -85,B 0,C 180,E1 -5162.945,E2 -5162.945} C_VEL
LIN {X 0,Y 516.886,Z 653.89,A -85,B 0,C 180,E1 -5165.778,E2 -5165.778} C_VEL
LIN {X 0,Y 516.877,Z 653.909,A -85,B 0,C 180,E1 -5168.715,E2 -5168.715} C_VEL
LIN {X 0,Y 516.91,Z 653.91,A -85,B 0,C 180,E1 -5171.774,E2 -5171.774} C_VEL
LIN {X 0,Y 516.916,Z 653.897,A -85,B 0,C 180,E1 -5175.009,E2 -5175.009} C_VEL
LIN {X 0,Y 516.923,Z 653.894,A -85,B 0,C 180,E1 -5178.396,E2 -5178.396} C_VEL
LIN {X 0,Y 516.899,Z 653.908,A -85,B 0,C 180,E1 -5181.286,E2 -5181.286} C_VEL
LIN {X 0,Y 516.884,Z 653.901,A -85,B 0,C 180,E1 -5184.221,E2 -5184.221} C_VEL
LIN {X 0,Y 516.89,Z 653.906,A -85,B 0,C 180,E1 -5187.053,E2 -5187.053} C_VEL
LIN {X 0,Y 516.893,Z 653.904,A -85,B 0,C 180,E1 -5189.796,E2 -5189.796} C_VEL
LIN {X 0,Y 516.921,Z 653.897,A -85,B 0,C 180,E1 -5192.467,E2 -5192.467} C_VEL
LIN {X 0,Y 516.902,Z 653.906,A -85,B 0,C 180,E1 -5195.071,E2 -5195.071} C_VEL
LIN {X 0,Y 516.877,Z 653.912,A -85,B 0,C 180,E1 -5198.462,E2 -5198.462} C_VEL
LIN {X 0,Y 516.895,Z 653.906,A -85,B 0,C 180,E1 -5200.954,E2 -5200.954} C_VEL
LIN {X 0,Y 516.908,Z 653.904,A -85,B 0,C 180,E1 -5203.41,E2 -5203.41} C_VEL
LIN {X 0,Y 516.885,Z 653.905,A -85,B 0,C 180,E1 -5205.833,E2 -5205.833} C_VEL
LIN {X 0,Y 516.993,Z 653.891,A -85,B 0,C 180,E1 -5208.234,E2 -5208.234} C_VEL
LIN {X 0,Y 516.963,Z 653.893,A -85,B 0,C 180,E1 -5211.399,E2 -5211.399} C_VEL
LIN {X 0,Y 517.053,Z 653.886,A -85,B 0,C 180,E1 -5214.54,E2 -5214.54} C_VEL
LIN {X 0,Y 517.074,Z 653.884,A -85,B 0,C 180,E1 -5217.663,E2 -5217.663} C_VEL
LIN {X 0,Y 517.086,Z 653.883,A -85,B 0,C 180,E1 -5220.779,E2 -5220.779} C_VEL
LIN {X 0,Y 517.008,Z 653.888,A -85,B 0,C 180,E1 -5223.117,E2 -5223.117} C_VEL
LIN {X 0,Y 517.005,Z 653.891,A -85,B 0,C 180,E1 -5226.243,E2 -5226.243} C_VEL
LIN {X 0,Y 516.948,Z 653.9,A -85,B 0,C 180,E1 -5229.389,E2 -5229.389} C_VEL
LIN {X 0,Y 516.945,Z 653.903,A -85,B 0,C 180,E1 -5231.81,E2 -5231.81} C_VEL
LIN {X 0,Y 516.932,Z 653.901,A -85,B 0,C 180,E1 -5235.146,E2 -5235.146} C_VEL
LIN {X 0,Y 516.914,Z 653.907,A -85,B 0,C 180,E1 -5238.222,E2 -5238.222} C_VEL
LIN {X 0,Y 516.905,Z 653.905,A -85,B 0,C 180,E1 -5240.701,E2 -5240.701} C_VEL
LIN {X 0,Y 516.884,Z 653.905,A -85,B 0,C 180,E1 -5243.222,E2 -5243.222} C_VEL
LIN {X 0,Y 516.934,Z 653.906,A -85,B 0,C 180,E1 -5246.197,E2 -5246.197} C_VEL
LIN {X 0,Y 516.925,Z 653.889,A -85,B 0,C 180,E1 -5249.304,E2 -5249.304} C_VEL
LIN {X 0,Y 516.891,Z 653.914,A -85,B 0,C 180,E1 -5252.545,E2 -5252.545} C_VEL
LIN {X 0,Y 516.873,Z 653.896,A -85,B 0,C 180,E1 -5255.333,E2 -5255.333} C_VEL
LIN {X 0,Y 516.872,Z 653.905,A -85,B 0,C 180,E1 -5257.944,E2 -5257.944} C_VEL
LIN {X 0,Y 516.899,Z 653.911,A -85,B 0,C 180,E1 -5260.74,E2 -5260.74} C_VEL
LIN {X 0,Y 516.874,Z 653.91,A -85,B 0,C 180,E1 -5263.903,E2 -5263.903} C_VEL
LIN {X 0,Y 516.873,Z 653.909,A -85,B 0,C 180,E1 -5266.107,E2 -5266.107} C_VEL
LIN {X 0,Y 516.896,Z 653.914,A -85,B 0,C 180,E1 -5269.261,E2 -5269.261} C_VEL
LIN {X 0,Y 516.893,Z 653.906,A -85,B 0,C 180,E1 -5270.31,E2 -5270.31} C_VEL
LIN {X 0,Y 516.213,Z 653.995,A -85,B 0,C 180,E1 -5270.96,E2 -5270.96} C_VEL
LIN {X 0,Y 513.36,Z 654.356,A -85,B 0,C 180,E1 -5272.015,E2 -5272.015} C_VEL
LIN {X 0,Y 510.952,Z 654.659,A -85,B 0,C 180,E1 -5272.866,E2 -5272.866} C_VEL
LIN {X 0,Y 509.913,Z 654.785,A -85,B 0,C 180,E1 -5273.522,E2 -5273.522} C_VEL
LIN {X 0,Y 509.825,Z 654.793,A -85,B 0,C 180,E1 -5273.744,E2 -5273.744} C_VEL
LIN {X 0,Y 509.855,Z 654.784,A -85,B 0,C 180,E1 -5276.54,E2 -5276.54} C_VEL
LIN {X 0,Y 509.844,Z 654.789,A -85,B 0,C 180,E1 -5279.335,E2 -5279.335} C_VEL
LIN {X 0,Y 509.889,Z 654.785,A -85,B 0,C 180,E1 -5282.055,E2 -5282.055} C_VEL
LIN {X 0,Y 509.871,Z 654.783,A -85,B 0,C 180,E1 -5284.704,E2 -5284.704} C_VEL
LIN {X 0,Y 509.831,Z 654.789,A -85,B 0,C 180,E1 -5287.455,E2 -5287.455} C_VEL
LIN {X 0,Y 509.912,Z 654.781,A -85,B 0,C 180,E1 -5289.845,E2 -5289.845} C_VEL
LIN {X 0,Y 509.88,Z 654.781,A -85,B 0,C 180,E1 -5293.175,E2 -5293.175} C_VEL
LIN {X 0,Y 509.86,Z 654.785,A -85,B 0,C 180,E1 -5295.634,E2 -5295.634} C_VEL
LIN {X 0,Y 509.909,Z 654.783,A -85,B 0,C 180,E1 -5298.875,E2 -5298.875} C_VEL
LIN {X 0,Y 509.948,Z 654.775,A -85,B 0,C 180,E1 -5302.079,E2 -5302.079} C_VEL
LIN {X 0,Y 509.978,Z 654.773,A -85,B 0,C 180,E1 -5304.464,E2 -5304.464} C_VEL
LIN {X 0,Y 510.052,Z 654.76,A -85,B 0,C 180,E1 -5307.631,E2 -5307.631} C_VEL
LIN {X 0,Y 510.06,Z 654.764,A -85,B 0,C 180,E1 -5310.789,E2 -5310.789} C_VEL
LIN {X 0,Y 509.953,Z 654.778,A -85,B 0,C 180,E1 -5313.16,E2 -5313.16} C_VEL
LIN {X 0,Y 509.975,Z 654.77,A -85,B 0,C 180,E1 -5316.329,E2 -5316.329} C_VEL
LIN {X 0,Y 509.912,Z 654.779,A -85,B 0,C 180,E1 -5318.72,E2 -5318.72} C_VEL
LIN {X 0,Y 509.9,Z 654.782,A -85,B 0,C 180,E1 -5321.931,E2 -5321.931} C_VEL
LIN {X 0,Y 509.889,Z 654.785,A -85,B 0,C 180,E1 -5325.242,E2 -5325.242} C_VEL
LIN {X 0,Y 509.884,Z 654.786,A -85,B 0,C 180,E1 -5328.001,E2 -5328.001} C_VEL
LIN {X 0,Y 509.845,Z 654.786,A -85,B 0,C 180,E1 -5331.001,E2 -5331.001} C_VEL
LIN {X 0,Y 509.831,Z 654.791,A -85,B 0,C 180,E1 -5333.563,E2 -5333.563} C_VEL
LIN {X 0,Y 509.906,Z 654.783,A -85,B 0,C 180,E1 -5336.378,E2 -5336.378} C_VEL
LIN {X 0,Y 509.88,Z 654.782,A -85,B 0,C 180,E1 -5338.843,E2 -5338.843} C_VEL
LIN {X 0,Y 509.82,Z 654.789,A -85,B 0,C 180,E1 -5341.589,E2 -5341.589} C_VEL
LIN {X 0,Y 509.846,Z 654.792,A -85,B 0,C 180,E1 -5344.413,E2 -5344.413} C_VEL
LIN {X 0,Y 509.812,Z 654.79,A -85,B 0,C 180,E1 -5347.34,E2 -5347.34} C_VEL
LIN {X 0,Y 509.853,Z 654.789,A -85,B 0,C 180,E1 -5350.379,E2 -5350.379} C_VEL
LIN {X 0,Y 509.815,Z 654.793,A -85,B 0,C 180,E1 -5353.062,E2 -5353.062} C_VEL
LIN {X 0,Y 509.822,Z 654.788,A -85,B 0,C 180,E1 -5355.792,E2 -5355.792} C_VEL
LIN {X 0,Y 509.862,Z 654.787,A -85,B 0,C 180,E1 -5358.576,E2 -5358.576} C_VEL
LIN {X 0,Y 509.846,Z 654.781,A -85,B 0,C 180,E1 -5361.785,E2 -5361.785} C_VEL
LIN {X 0,Y 509.836,Z 654.772,A -85,B 0,C 180,E1 -5364.623,E2 -5364.623} C_VEL
LIN {X 0,Y 509.856,Z 654.789,A -85,B 0,C 180,E1 -5367.481,E2 -5367.481} C_VEL
LIN {X 0,Y 509.871,Z 654.767,A -85,B 0,C 180,E1 -5370.269,E2 -5370.269} C_VEL
LIN {X 0,Y 509.876,Z 654.77,A -85,B 0,C 180,E1 -5372.944,E2 -5372.944} C_VEL
LIN {X 0,Y 509.865,Z 654.79,A -85,B 0,C 180,E1 -5375.574,E2 -5375.574} C_VEL
LIN {X 0,Y 509.842,Z 654.786,A -85,B 0,C 180,E1 -5378.15,E2 -5378.15} C_VEL
LIN {X 0,Y 509.854,Z 654.782,A -85,B 0,C 180,E1 -5380.682,E2 -5380.682} C_VEL
LIN {X 0,Y 509.876,Z 654.776,A -85,B 0,C 180,E1 -5383.175,E2 -5383.175} C_VEL
LIN {X 0,Y 509.853,Z 654.785,A -85,B 0,C 180,E1 -5385.634,E2 -5385.634} C_VEL
LIN {X 0,Y 509.907,Z 654.776,A -85,B 0,C 180,E1 -5388.875,E2 -5388.875} C_VEL
LIN {X 0,Y 509.941,Z 654.772,A -85,B 0,C 180,E1 -5392.079,E2 -5392.079} C_VEL
LIN {X 0,Y 510,Z 654.773,A -85,B 0,C 180,E1 -5394.465,E2 -5394.465} C_VEL
LIN {X 0,Y 510.045,Z 654.751,A -85,B 0,C 180,E1 -5397.631,E2 -5397.631} C_VEL
LIN {X 0,Y 510.056,Z 654.763,A -85,B 0,C 180,E1 -5400.79,E2 -5400.79} C_VEL
LIN {X 0,Y 509.95,Z 654.771,A -85,B 0,C 180,E1 -5403.16,E2 -5403.16} C_VEL
LIN {X 0,Y 509.972,Z 654.769,A -85,B 0,C 180,E1 -5406.33,E2 -5406.33} C_VEL
LIN {X 0,Y 509.909,Z 654.773,A -85,B 0,C 180,E1 -5408.72,E2 -5408.72} C_VEL
LIN {X 0,Y 509.94,Z 654.768,A -85,B 0,C 180,E1 -5411.931,E2 -5411.931} C_VEL
LIN {X 0,Y 509.883,Z 654.787,A -85,B 0,C 180,E1 -5415.242,E2 -5415.242} C_VEL
LIN {X 0,Y 509.878,Z 654.777,A -85,B 0,C 180,E1 -5418.001,E2 -5418.001} C_VEL
LIN {X 0,Y 509.841,Z 654.787,A -85,B 0,C 180,E1 -5421.002,E2 -5421.002} C_VEL
LIN {X 0,Y 509.827,Z 654.79,A -85,B 0,C 180,E1 -5423.564,E2 -5423.564} C_VEL
LIN {X 0,Y 509.904,Z 654.772,A -85,B 0,C 180,E1 -5426.38,E2 -5426.38} C_VEL
LIN {X 0,Y 509.877,Z 654.757,A -85,B 0,C 180,E1 -5428.844,E2 -5428.844} C_VEL
LIN {X 0,Y 509.818,Z 654.788,A -85,B 0,C 180,E1 -5431.59,E2 -5431.59} C_VEL
LIN {X 0,Y 509.847,Z 654.779,A -85,B 0,C 180,E1 -5434.414,E2 -5434.414} C_VEL
LIN {X 0,Y 509.812,Z 654.785,A -85,B 0,C 180,E1 -5437.341,E2 -5437.341} C_VEL
LIN {X 0,Y 509.872,Z 654.777,A -85,B 0,C 180,E1 -5440.379,E2 -5440.379} C_VEL
LIN {X 0,Y 509.834,Z 654.788,A -85,B 0,C 180,E1 -5443.065,E2 -5443.065} C_VEL
LIN {X 0,Y 509.824,Z 654.779,A -85,B 0,C 180,E1 -5445.793,E2 -5445.793} C_VEL
LIN {X 0,Y 509.853,Z 654.785,A -85,B 0,C 180,E1 -5448.576,E2 -5448.576} C_VEL
LIN {X 0,Y 509.846,Z 654.783,A -85,B 0,C 180,E1 -5451.787,E2 -5451.787} C_VEL
LIN {X 0,Y 509.841,Z 654.773,A -85,B 0,C 180,E1 -5454.624,E2 -5454.624} C_VEL
LIN {X 0,Y 509.886,Z 654.925,A -85,B 0,C 180,E1 -5456.919,E2 -5456.919} C_VEL
LIN {X 0,Y 513.333,Z 668.731,A -85,B 0,C 180,E1 -5459.338,E2 -5459.338} C_VEL
LIN {X 0,Y 514.055,Z 673.21,A -85,B 0,C 180,E1 -5460.066,E2 -5460.066} C_VEL
LIN {X 0,Y 513.312,Z 690.522,A -85,B 0,C 180,E1 -5462.639,E2 -5462.639} C_VEL
LIN {X 0,Y 513.24,Z 695.312,A -85,B 0,C 180,E1 -5463.308,E2 -5463.308} C_VEL
LIN {X 0,Y 518.061,Z 715.023,A -85,B 0,C 180,E1 -5463.886,E2 -5463.886} C_VEL
LIN {X 0,Y 516.393,Z 896.807,A -85,B 0,C 180,E1 -5466.542,E2 -5466.542} C_VEL
LIN {X 0,Y 516.015,Z 909.945,A -85,B 0,C 180,E1 -5466.816,E2 -5466.816} C_VEL
LIN {X 0,Y 515.684,Z 923.057,A -85,B 0,C 180,E1 -5467.198,E2 -5467.198} C_VEL
LIN {X 0,Y 515.22,Z 935.676,A -85,B 0,C 180,E1 -5467.663,E2 -5467.663} C_VEL
LIN {X 0,Y 514.778,Z 947.243,A -85,B 0,C 180,E1 -5468.182,E2 -5468.182} C_VEL
LIN {X 0,Y 514.187,Z 960.076,A -85,B 0,C 180,E1 -5468.87,E2 -5468.87} C_VEL
LIN {X 0,Y 513.542,Z 972.824,A -85,B 0,C 180,E1 -5469.68,E2 -5469.68} C_VEL
LIN {X 0,Y 512.95,Z 983.828,A -85,B 0,C 180,E1 -5470.491,E2 -5470.491} C_VEL
LIN {X 0,Y 512.351,Z 995.009,A -85,B 0,C 180,E1 -5471.443,E2 -5471.443} C_VEL
LIN {X 0,Y 511.794,Z 1005.03,A -85,B 0,C 180,E1 -5472.416,E2 -5472.416} C_VEL
LIN {X 0,Y 511.308,Z 1014.244,A -85,B 0,C 180,E1 -5473.429,E2 -5473.429} C_VEL
LIN {X 0,Y 510.794,Z 1024.198,A -85,B 0,C 180,E1 -5474.682,E2 -5474.682} C_VEL
LIN {X 0,Y 510.303,Z 1033.639,A -85,B 0,C 180,E1 -5476.054,E2 -5476.054} C_VEL
LIN {X 0,Y 509.979,Z 1040.896,A -85,B 0,C 180,E1 -5477.262,E2 -5477.262} C_VEL
LIN {X 0,Y 509.776,Z 1047.425,A -85,B 0,C 180,E1 -5478.503,E2 -5478.503} C_VEL
LIN {X 0,Y 509.487,Z 1054.447,A -85,B 0,C 180,E1 -5480.071,E2 -5480.071} C_VEL
